//     PlcTask Inputs/GVL_iXlinker.EtherCAT_Master_EPPxxxx.Beckhoff_EPP6xxx.Beckhoff_EPP6xxxEK1122.A_0009_EPP6228_0022_0016.Module_1_DeviceState_Inputs_Device.DeviceState_Inputs_Device.Device_State <-> Module 1 (DeviceState Inputs Device)/DeviceState Inputs Device/Device State
//     PlcTask Inputs/GVL_iXlinker.EtherCAT_Master_EPPxxxx.Beckhoff_EPP6xxx.Beckhoff_EPP6xxxEK1122.A_0009_EPP6228_0022_0016.Module_2_DeviceState_Inputs.DeviceState_Inputs.State_Ch1 <-> Module 2 (DeviceState Inputs)/DeviceState Inputs/State Ch1
//     PlcTask Inputs/GVL_iXlinker.EtherCAT_Master_EPPxxxx.Beckhoff_EPP6xxx.Beckhoff_EPP6xxxEK1122.A_0009_EPP6228_0022_0016.Module_2_DeviceState_Inputs.DeviceState_Inputs.State_Ch2 <-> Module 2 (DeviceState Inputs)/DeviceState Inputs/State Ch2
//     PlcTask Inputs/GVL_iXlinker.EtherCAT_Master_EPPxxxx.Beckhoff_EPP6xxx.Beckhoff_EPP6xxxEK1122.A_0009_EPP6228_0022_0016.Module_2_DeviceState_Inputs.DeviceState_Inputs.State_Ch3 <-> Module 2 (DeviceState Inputs)/DeviceState Inputs/State Ch3
//     PlcTask Inputs/GVL_iXlinker.EtherCAT_Master_EPPxxxx.Beckhoff_EPP6xxx.Beckhoff_EPP6xxxEK1122.A_0009_EPP6228_0022_0016.Module_2_DeviceState_Inputs.DeviceState_Inputs.State_Ch4 <-> Module 2 (DeviceState Inputs)/DeviceState Inputs/State Ch4
//     PlcTask Inputs/GVL_iXlinker.EtherCAT_Master_EPPxxxx.Beckhoff_EPP6xxx.Beckhoff_EPP6xxxEK1122.A_0009_EPP6228_0022_0016.Module_2_DeviceState_Inputs.DeviceState_Inputs.State_Ch5 <-> Module 2 (DeviceState Inputs)/DeviceState Inputs/State Ch5
//     PlcTask Inputs/GVL_iXlinker.EtherCAT_Master_EPPxxxx.Beckhoff_EPP6xxx.Beckhoff_EPP6xxxEK1122.A_0009_EPP6228_0022_0016.Module_2_DeviceState_Inputs.DeviceState_Inputs.State_Ch6 <-> Module 2 (DeviceState Inputs)/DeviceState Inputs/State Ch6
//     PlcTask Inputs/GVL_iXlinker.EtherCAT_Master_EPPxxxx.Beckhoff_EPP6xxx.Beckhoff_EPP6xxxEK1122.A_0009_EPP6228_0022_0016.Module_2_DeviceState_Inputs.DeviceState_Inputs.State_Ch7 <-> Module 2 (DeviceState Inputs)/DeviceState Inputs/State Ch7
//     PlcTask Inputs/GVL_iXlinker.EtherCAT_Master_EPPxxxx.Beckhoff_EPP6xxx.Beckhoff_EPP6xxxEK1122.A_0009_EPP6228_0022_0016.Module_2_DeviceState_Inputs.DeviceState_Inputs.State_Ch8 <-> Module 2 (DeviceState Inputs)/DeviceState Inputs/State Ch8
//     PlcTask Inputs/GVL_iXlinker.EtherCAT_Master_EPPxxxx.Beckhoff_EPP6xxx.Beckhoff_EPP6xxxEK1122.A_0009_EPP6228_0022_0016.Module_11_Digital_Inputs.Digital_Inputs.Pin2_Ch1 <-> Module 11 (Digital Inputs)/Digital Inputs/Pin2 Ch1
//     PlcTask Inputs/GVL_iXlinker.EtherCAT_Master_EPPxxxx.Beckhoff_EPP6xxx.Beckhoff_EPP6xxxEK1122.A_0009_EPP6228_0022_0016.Module_11_Digital_Inputs.Digital_Inputs.Pin2_Ch2 <-> Module 11 (Digital Inputs)/Digital Inputs/Pin2 Ch2
//     PlcTask Inputs/GVL_iXlinker.EtherCAT_Master_EPPxxxx.Beckhoff_EPP6xxx.Beckhoff_EPP6xxxEK1122.A_0009_EPP6228_0022_0016.Module_11_Digital_Inputs.Digital_Inputs.Pin2_Ch3 <-> Module 11 (Digital Inputs)/Digital Inputs/Pin2 Ch3
//     PlcTask Inputs/GVL_iXlinker.EtherCAT_Master_EPPxxxx.Beckhoff_EPP6xxx.Beckhoff_EPP6xxxEK1122.A_0009_EPP6228_0022_0016.Module_11_Digital_Inputs.Digital_Inputs.Pin2_Ch4 <-> Module 11 (Digital Inputs)/Digital Inputs/Pin2 Ch4
//     PlcTask Inputs/GVL_iXlinker.EtherCAT_Master_EPPxxxx.Beckhoff_EPP6xxx.Beckhoff_EPP6xxxEK1122.A_0009_EPP6228_0022_0016.Module_11_Digital_Inputs.Digital_Inputs.Pin2_Ch5 <-> Module 11 (Digital Inputs)/Digital Inputs/Pin2 Ch5
//     PlcTask Inputs/GVL_iXlinker.EtherCAT_Master_EPPxxxx.Beckhoff_EPP6xxx.Beckhoff_EPP6xxxEK1122.A_0009_EPP6228_0022_0016.Module_11_Digital_Inputs.Digital_Inputs.Pin2_Ch6 <-> Module 11 (Digital Inputs)/Digital Inputs/Pin2 Ch6
//     PlcTask Inputs/GVL_iXlinker.EtherCAT_Master_EPPxxxx.Beckhoff_EPP6xxx.Beckhoff_EPP6xxxEK1122.A_0009_EPP6228_0022_0016.Module_11_Digital_Inputs.Digital_Inputs.Pin2_Ch7 <-> Module 11 (Digital Inputs)/Digital Inputs/Pin2 Ch7
//     PlcTask Inputs/GVL_iXlinker.EtherCAT_Master_EPPxxxx.Beckhoff_EPP6xxx.Beckhoff_EPP6xxxEK1122.A_0009_EPP6228_0022_0016.Module_11_Digital_Inputs.Digital_Inputs.Pin2_Ch8 <-> Module 11 (Digital Inputs)/Digital Inputs/Pin2 Ch8
//     PlcTask Inputs/GVL_iXlinker.EtherCAT_Master_EPPxxxx.Beckhoff_EPP6xxx.Beckhoff_EPP6xxxEK1122.A_0009_EPP6228_0022_0016.WcState.WcState <-> WcState/WcState
//     PlcTask Inputs/GVL_iXlinker.EtherCAT_Master_EPPxxxx.Beckhoff_EPP6xxx.Beckhoff_EPP6xxxEK1122.A_0009_EPP6228_0022_0016.WcState.InputToggle <-> WcState/InputToggle
//     PlcTask Inputs/GVL_iXlinker.EtherCAT_Master_EPPxxxx.Beckhoff_EPP6xxx.Beckhoff_EPP6xxxEK1122.A_0009_EPP6228_0022_0016.InfoData.AdsAddr <-> InfoData/AdsAddr
//     PlcTask Inputs/GVL_iXlinker.EtherCAT_Master_EPPxxxx.Beckhoff_EPP6xxx.Beckhoff_EPP6xxxEK1122.A_0009_EPP6228_0022_0016.InfoData.AoeNetId <-> InfoData/AoeNetId
//     PlcTask Inputs/GVL_iXlinker.EtherCAT_Master_EPPxxxx.Beckhoff_EPP6xxx.Beckhoff_EPP6xxxEK1122.A_0009_EPP6228_0022_0016.InfoData.State <-> InfoData/State
//   PLC/PLC Instance <-> EtherCAT Master EPPxxxx/Beckhoff EPP7xxx
//     PlcTask Inputs/GVL_iXlinker.EtherCAT_Master_EPPxxxx.Beckhoff_EPP7xxx.InfoData.State <-> InfoData/State
//   PLC/PLC Instance <-> EtherCAT Master EPPxxxx/Beckhoff EPP7xxx/Beckhoff EPP7xxxEK1122
//     PlcTask Inputs/GVL_iXlinker.EtherCAT_Master_EPPxxxx.Beckhoff_EPP7xxx.Beckhoff_EPP7xxxEK1122.InfoData.State <-> InfoData/State
//   PLC/PLC Instance <-> EtherCAT Master EPPxxxx/Beckhoff EPP7xxx/Beckhoff EPP7xxxEK1122/Beckhoff EPP7xxxsub EK1100
//     PlcTask Inputs/GVL_iXlinker.EtherCAT_Master_EPPxxxx.Beckhoff_EPP7xxx.Beckhoff_EPP7xxxEK1122.Beckhoff_EPP7xxxsub_EK1100.InfoData.State <-> InfoData/State
//   PLC/PLC Instance <-> EtherCAT Master EPPxxxx/Beckhoff EPP7xxx/Beckhoff EPP7xxxEK1122/A_0001(EPP7041-1002-0016)
//     PlcTask Inputs/GVL_iXlinker.EtherCAT_Master_EPPxxxx.Beckhoff_EPP7xxx.Beckhoff_EPP7xxxEK1122.A_0001_EPP7041_1002_0016.ENC_Status_compact.Status/Latch_C_valid <-> ENC Status compact/Status/Latch C valid
//     PlcTask Inputs/GVL_iXlinker.EtherCAT_Master_EPPxxxx.Beckhoff_EPP7xxx.Beckhoff_EPP7xxxEK1122.A_0001_EPP7041_1002_0016.ENC_Status_compact.Status/Latch_extern_valid <-> ENC Status compact/Status/Latch extern valid
//     PlcTask Inputs/GVL_iXlinker.EtherCAT_Master_EPPxxxx.Beckhoff_EPP7xxx.Beckhoff_EPP7xxxEK1122.A_0001_EPP7041_1002_0016.ENC_Status_compact.Status/Set_counter_done <-> ENC Status compact/Status/Set counter done
//     PlcTask Inputs/GVL_iXlinker.EtherCAT_Master_EPPxxxx.Beckhoff_EPP7xxx.Beckhoff_EPP7xxxEK1122.A_0001_EPP7041_1002_0016.ENC_Status_compact.Status/Counter_underflow <-> ENC Status compact/Status/Counter underflow
//     PlcTask Inputs/GVL_iXlinker.EtherCAT_Master_EPPxxxx.Beckhoff_EPP7xxx.Beckhoff_EPP7xxxEK1122.A_0001_EPP7041_1002_0016.ENC_Status_compact.Status/Counter_overflow <-> ENC Status compact/Status/Counter overflow
//     PlcTask Inputs/GVL_iXlinker.EtherCAT_Master_EPPxxxx.Beckhoff_EPP7xxx.Beckhoff_EPP7xxxEK1122.A_0001_EPP7041_1002_0016.ENC_Status_compact.Status/Extrapolation_stall <-> ENC Status compact/Status/Extrapolation stall
//     PlcTask Inputs/GVL_iXlinker.EtherCAT_Master_EPPxxxx.Beckhoff_EPP7xxx.Beckhoff_EPP7xxxEK1122.A_0001_EPP7041_1002_0016.ENC_Status_compact.Status/Status_of_input_A <-> ENC Status compact/Status/Status of input A
//     PlcTask Inputs/GVL_iXlinker.EtherCAT_Master_EPPxxxx.Beckhoff_EPP7xxx.Beckhoff_EPP7xxxEK1122.A_0001_EPP7041_1002_0016.ENC_Status_compact.Status/Status_of_input_B <-> ENC Status compact/Status/Status of input B
//     PlcTask Inputs/GVL_iXlinker.EtherCAT_Master_EPPxxxx.Beckhoff_EPP7xxx.Beckhoff_EPP7xxxEK1122.A_0001_EPP7041_1002_0016.ENC_Status_compact.Status/Status_of_input_C <-> ENC Status compact/Status/Status of input C
//     PlcTask Inputs/GVL_iXlinker.EtherCAT_Master_EPPxxxx.Beckhoff_EPP7xxx.Beckhoff_EPP7xxxEK1122.A_0001_EPP7041_1002_0016.ENC_Status_compact.Status/Status_of_extern_latch <-> ENC Status compact/Status/Status of extern latch
//     PlcTask Inputs/GVL_iXlinker.EtherCAT_Master_EPPxxxx.Beckhoff_EPP7xxx.Beckhoff_EPP7xxxEK1122.A_0001_EPP7041_1002_0016.ENC_Status_compact.Status/Sync_error <-> ENC Status compact/Status/Sync error
//     PlcTask Inputs/GVL_iXlinker.EtherCAT_Master_EPPxxxx.Beckhoff_EPP7xxx.Beckhoff_EPP7xxxEK1122.A_0001_EPP7041_1002_0016.ENC_Status_compact.Status/TxPDO_Toggle <-> ENC Status compact/Status/TxPDO Toggle
//     PlcTask Inputs/GVL_iXlinker.EtherCAT_Master_EPPxxxx.Beckhoff_EPP7xxx.Beckhoff_EPP7xxxEK1122.A_0001_EPP7041_1002_0016.ENC_Status_compact.Counter_value <-> ENC Status compact/Counter value
//     PlcTask Inputs/GVL_iXlinker.EtherCAT_Master_EPPxxxx.Beckhoff_EPP7xxx.Beckhoff_EPP7xxxEK1122.A_0001_EPP7041_1002_0016.ENC_Status_compact.Latch_value <-> ENC Status compact/Latch value
//     PlcTask Inputs/GVL_iXlinker.EtherCAT_Master_EPPxxxx.Beckhoff_EPP7xxx.Beckhoff_EPP7xxxEK1122.A_0001_EPP7041_1002_0016.STM_Status.Status/Ready_to_enable <-> STM Status/Status/Ready to enable
//     PlcTask Inputs/GVL_iXlinker.EtherCAT_Master_EPPxxxx.Beckhoff_EPP7xxx.Beckhoff_EPP7xxxEK1122.A_0001_EPP7041_1002_0016.STM_Status.Status/Ready <-> STM Status/Status/Ready
//     PlcTask Inputs/GVL_iXlinker.EtherCAT_Master_EPPxxxx.Beckhoff_EPP7xxx.Beckhoff_EPP7xxxEK1122.A_0001_EPP7041_1002_0016.STM_Status.Status/Warning <-> STM Status/Status/Warning
//     PlcTask Inputs/GVL_iXlinker.EtherCAT_Master_EPPxxxx.Beckhoff_EPP7xxx.Beckhoff_EPP7xxxEK1122.A_0001_EPP7041_1002_0016.STM_Status.Status/Error <-> STM Status/Status/Error
//     PlcTask Inputs/GVL_iXlinker.EtherCAT_Master_EPPxxxx.Beckhoff_EPP7xxx.Beckhoff_EPP7xxxEK1122.A_0001_EPP7041_1002_0016.STM_Status.Status/Moving_positive <-> STM Status/Status/Moving positive
//     PlcTask Inputs/GVL_iXlinker.EtherCAT_Master_EPPxxxx.Beckhoff_EPP7xxx.Beckhoff_EPP7xxxEK1122.A_0001_EPP7041_1002_0016.STM_Status.Status/Moving_negative <-> STM Status/Status/Moving negative
//     PlcTask Inputs/GVL_iXlinker.EtherCAT_Master_EPPxxxx.Beckhoff_EPP7xxx.Beckhoff_EPP7xxxEK1122.A_0001_EPP7041_1002_0016.STM_Status.Status/Torque_reduced <-> STM Status/Status/Torque reduced
//     PlcTask Inputs/GVL_iXlinker.EtherCAT_Master_EPPxxxx.Beckhoff_EPP7xxx.Beckhoff_EPP7xxxEK1122.A_0001_EPP7041_1002_0016.STM_Status.Status/Digital_input_1 <-> STM Status/Status/Digital input 1
//     PlcTask Inputs/GVL_iXlinker.EtherCAT_Master_EPPxxxx.Beckhoff_EPP7xxx.Beckhoff_EPP7xxxEK1122.A_0001_EPP7041_1002_0016.STM_Status.Status/Digital_input_2 <-> STM Status/Status/Digital input 2
//     PlcTask Inputs/GVL_iXlinker.EtherCAT_Master_EPPxxxx.Beckhoff_EPP7xxx.Beckhoff_EPP7xxxEK1122.A_0001_EPP7041_1002_0016.STM_Status.Status/Sync_error <-> STM Status/Status/Sync error
//     PlcTask Inputs/GVL_iXlinker.EtherCAT_Master_EPPxxxx.Beckhoff_EPP7xxx.Beckhoff_EPP7xxxEK1122.A_0001_EPP7041_1002_0016.STM_Status.Status/TxPDO_Toggle <-> STM Status/Status/TxPDO Toggle
//     PlcTask Outputs/GVL_iXlinker.EtherCAT_Master_EPPxxxx.Beckhoff_EPP7xxx.Beckhoff_EPP7xxxEK1122.A_0001_EPP7041_1002_0016.ENC_Control_compact.Control/Enable_latch_C <-> ENC Control compact/Control/Enable latch C
//     PlcTask Outputs/GVL_iXlinker.EtherCAT_Master_EPPxxxx.Beckhoff_EPP7xxx.Beckhoff_EPP7xxxEK1122.A_0001_EPP7041_1002_0016.ENC_Control_compact.Control/Enable_latch_extern_on_positive_edge <-> ENC Control compact/Control/Enable latch extern on positive edge
//     PlcTask Outputs/GVL_iXlinker.EtherCAT_Master_EPPxxxx.Beckhoff_EPP7xxx.Beckhoff_EPP7xxxEK1122.A_0001_EPP7041_1002_0016.ENC_Control_compact.Control/Set_counter <-> ENC Control compact/Control/Set counter
//     PlcTask Outputs/GVL_iXlinker.EtherCAT_Master_EPPxxxx.Beckhoff_EPP7xxx.Beckhoff_EPP7xxxEK1122.A_0001_EPP7041_1002_0016.ENC_Control_compact.Control/Enable_latch_extern_on_negative_edge <-> ENC Control compact/Control/Enable latch extern on negative edge
//     PlcTask Outputs/GVL_iXlinker.EtherCAT_Master_EPPxxxx.Beckhoff_EPP7xxx.Beckhoff_EPP7xxxEK1122.A_0001_EPP7041_1002_0016.ENC_Control_compact.Set_counter_value <-> ENC Control compact/Set counter value
//     PlcTask Outputs/GVL_iXlinker.EtherCAT_Master_EPPxxxx.Beckhoff_EPP7xxx.Beckhoff_EPP7xxxEK1122.A_0001_EPP7041_1002_0016.STM_Control.Control/Enable <-> STM Control/Control/Enable
//     PlcTask Outputs/GVL_iXlinker.EtherCAT_Master_EPPxxxx.Beckhoff_EPP7xxx.Beckhoff_EPP7xxxEK1122.A_0001_EPP7041_1002_0016.STM_Control.Control/Reset <-> STM Control/Control/Reset
//     PlcTask Outputs/GVL_iXlinker.EtherCAT_Master_EPPxxxx.Beckhoff_EPP7xxx.Beckhoff_EPP7xxxEK1122.A_0001_EPP7041_1002_0016.STM_Control.Control/Reduce_torque <-> STM Control/Control/Reduce torque
//     PlcTask Outputs/GVL_iXlinker.EtherCAT_Master_EPPxxxx.Beckhoff_EPP7xxx.Beckhoff_EPP7xxxEK1122.A_0001_EPP7041_1002_0016.STM_Control.Control/Digital_output_1 <-> STM Control/Control/Digital output 1
//     PlcTask Outputs/GVL_iXlinker.EtherCAT_Master_EPPxxxx.Beckhoff_EPP7xxx.Beckhoff_EPP7xxxEK1122.A_0001_EPP7041_1002_0016.STM_Velocity.Velocity <-> STM Velocity/Velocity
//     PlcTask Inputs/GVL_iXlinker.EtherCAT_Master_EPPxxxx.Beckhoff_EPP7xxx.Beckhoff_EPP7xxxEK1122.A_0001_EPP7041_1002_0016.WcState.WcState <-> WcState/WcState
//     PlcTask Inputs/GVL_iXlinker.EtherCAT_Master_EPPxxxx.Beckhoff_EPP7xxx.Beckhoff_EPP7xxxEK1122.A_0001_EPP7041_1002_0016.WcState.InputToggle <-> WcState/InputToggle
//     PlcTask Inputs/GVL_iXlinker.EtherCAT_Master_EPPxxxx.Beckhoff_EPP7xxx.Beckhoff_EPP7xxxEK1122.A_0001_EPP7041_1002_0016.InfoData.AdsAddr <-> InfoData/AdsAddr
//     PlcTask Inputs/GVL_iXlinker.EtherCAT_Master_EPPxxxx.Beckhoff_EPP7xxx.Beckhoff_EPP7xxxEK1122.A_0001_EPP7041_1002_0016.InfoData.Chn0 <-> InfoData/Chn0
//     PlcTask Inputs/GVL_iXlinker.EtherCAT_Master_EPPxxxx.Beckhoff_EPP7xxx.Beckhoff_EPP7xxxEK1122.A_0001_EPP7041_1002_0016.InfoData.Chn1 <-> InfoData/Chn1
//     PlcTask Inputs/GVL_iXlinker.EtherCAT_Master_EPPxxxx.Beckhoff_EPP7xxx.Beckhoff_EPP7xxxEK1122.A_0001_EPP7041_1002_0016.InfoData.State <-> InfoData/State
//   PLC/PLC Instance <-> EtherCAT Master EPPxxxx/Beckhoff EPP7xxx/Beckhoff EPP7xxxEK1122/A_0002(EPP7041-1002-0017)
//     PlcTask Inputs/GVL_iXlinker.EtherCAT_Master_EPPxxxx.Beckhoff_EPP7xxx.Beckhoff_EPP7xxxEK1122.A_0002_EPP7041_1002_0017.ENC_Status_compact.Status/Latch_C_valid <-> ENC Status compact/Status/Latch C valid
//     PlcTask Inputs/GVL_iXlinker.EtherCAT_Master_EPPxxxx.Beckhoff_EPP7xxx.Beckhoff_EPP7xxxEK1122.A_0002_EPP7041_1002_0017.ENC_Status_compact.Status/Latch_extern_valid <-> ENC Status compact/Status/Latch extern valid
//     PlcTask Inputs/GVL_iXlinker.EtherCAT_Master_EPPxxxx.Beckhoff_EPP7xxx.Beckhoff_EPP7xxxEK1122.A_0002_EPP7041_1002_0017.ENC_Status_compact.Status/Set_counter_done <-> ENC Status compact/Status/Set counter done
//     PlcTask Inputs/GVL_iXlinker.EtherCAT_Master_EPPxxxx.Beckhoff_EPP7xxx.Beckhoff_EPP7xxxEK1122.A_0002_EPP7041_1002_0017.ENC_Status_compact.Status/Counter_underflow <-> ENC Status compact/Status/Counter underflow
//     PlcTask Inputs/GVL_iXlinker.EtherCAT_Master_EPPxxxx.Beckhoff_EPP7xxx.Beckhoff_EPP7xxxEK1122.A_0002_EPP7041_1002_0017.ENC_Status_compact.Status/Counter_overflow <-> ENC Status compact/Status/Counter overflow
//     PlcTask Inputs/GVL_iXlinker.EtherCAT_Master_EPPxxxx.Beckhoff_EPP7xxx.Beckhoff_EPP7xxxEK1122.A_0002_EPP7041_1002_0017.ENC_Status_compact.Status/Extrapolation_stall <-> ENC Status compact/Status/Extrapolation stall
//     PlcTask Inputs/GVL_iXlinker.EtherCAT_Master_EPPxxxx.Beckhoff_EPP7xxx.Beckhoff_EPP7xxxEK1122.A_0002_EPP7041_1002_0017.ENC_Status_compact.Status/Status_of_input_A <-> ENC Status compact/Status/Status of input A
//     PlcTask Inputs/GVL_iXlinker.EtherCAT_Master_EPPxxxx.Beckhoff_EPP7xxx.Beckhoff_EPP7xxxEK1122.A_0002_EPP7041_1002_0017.ENC_Status_compact.Status/Status_of_input_B <-> ENC Status compact/Status/Status of input B
//     PlcTask Inputs/GVL_iXlinker.EtherCAT_Master_EPPxxxx.Beckhoff_EPP7xxx.Beckhoff_EPP7xxxEK1122.A_0002_EPP7041_1002_0017.ENC_Status_compact.Status/Status_of_input_C <-> ENC Status compact/Status/Status of input C
//     PlcTask Inputs/GVL_iXlinker.EtherCAT_Master_EPPxxxx.Beckhoff_EPP7xxx.Beckhoff_EPP7xxxEK1122.A_0002_EPP7041_1002_0017.ENC_Status_compact.Status/Status_of_extern_latch <-> ENC Status compact/Status/Status of extern latch
//     PlcTask Inputs/GVL_iXlinker.EtherCAT_Master_EPPxxxx.Beckhoff_EPP7xxx.Beckhoff_EPP7xxxEK1122.A_0002_EPP7041_1002_0017.ENC_Status_compact.Status/Sync_error <-> ENC Status compact/Status/Sync error
//     PlcTask Inputs/GVL_iXlinker.EtherCAT_Master_EPPxxxx.Beckhoff_EPP7xxx.Beckhoff_EPP7xxxEK1122.A_0002_EPP7041_1002_0017.ENC_Status_compact.Status/TxPDO_Toggle <-> ENC Status compact/Status/TxPDO Toggle
//     PlcTask Inputs/GVL_iXlinker.EtherCAT_Master_EPPxxxx.Beckhoff_EPP7xxx.Beckhoff_EPP7xxxEK1122.A_0002_EPP7041_1002_0017.ENC_Status_compact.Counter_value <-> ENC Status compact/Counter value
//     PlcTask Inputs/GVL_iXlinker.EtherCAT_Master_EPPxxxx.Beckhoff_EPP7xxx.Beckhoff_EPP7xxxEK1122.A_0002_EPP7041_1002_0017.ENC_Status_compact.Latch_value <-> ENC Status compact/Latch value
//     PlcTask Inputs/GVL_iXlinker.EtherCAT_Master_EPPxxxx.Beckhoff_EPP7xxx.Beckhoff_EPP7xxxEK1122.A_0002_EPP7041_1002_0017.STM_Status.Status/Ready_to_enable <-> STM Status/Status/Ready to enable
//     PlcTask Inputs/GVL_iXlinker.EtherCAT_Master_EPPxxxx.Beckhoff_EPP7xxx.Beckhoff_EPP7xxxEK1122.A_0002_EPP7041_1002_0017.STM_Status.Status/Ready <-> STM Status/Status/Ready
//     PlcTask Inputs/GVL_iXlinker.EtherCAT_Master_EPPxxxx.Beckhoff_EPP7xxx.Beckhoff_EPP7xxxEK1122.A_0002_EPP7041_1002_0017.STM_Status.Status/Warning <-> STM Status/Status/Warning
//     PlcTask Inputs/GVL_iXlinker.EtherCAT_Master_EPPxxxx.Beckhoff_EPP7xxx.Beckhoff_EPP7xxxEK1122.A_0002_EPP7041_1002_0017.STM_Status.Status/Error <-> STM Status/Status/Error
//     PlcTask Inputs/GVL_iXlinker.EtherCAT_Master_EPPxxxx.Beckhoff_EPP7xxx.Beckhoff_EPP7xxxEK1122.A_0002_EPP7041_1002_0017.STM_Status.Status/Moving_positive <-> STM Status/Status/Moving positive
//     PlcTask Inputs/GVL_iXlinker.EtherCAT_Master_EPPxxxx.Beckhoff_EPP7xxx.Beckhoff_EPP7xxxEK1122.A_0002_EPP7041_1002_0017.STM_Status.Status/Moving_negative <-> STM Status/Status/Moving negative
//     PlcTask Inputs/GVL_iXlinker.EtherCAT_Master_EPPxxxx.Beckhoff_EPP7xxx.Beckhoff_EPP7xxxEK1122.A_0002_EPP7041_1002_0017.STM_Status.Status/Torque_reduced <-> STM Status/Status/Torque reduced
//     PlcTask Inputs/GVL_iXlinker.EtherCAT_Master_EPPxxxx.Beckhoff_EPP7xxx.Beckhoff_EPP7xxxEK1122.A_0002_EPP7041_1002_0017.STM_Status.Status/Digital_input_1 <-> STM Status/Status/Digital input 1
//     PlcTask Inputs/GVL_iXlinker.EtherCAT_Master_EPPxxxx.Beckhoff_EPP7xxx.Beckhoff_EPP7xxxEK1122.A_0002_EPP7041_1002_0017.STM_Status.Status/Digital_input_2 <-> STM Status/Status/Digital input 2
//     PlcTask Inputs/GVL_iXlinker.EtherCAT_Master_EPPxxxx.Beckhoff_EPP7xxx.Beckhoff_EPP7xxxEK1122.A_0002_EPP7041_1002_0017.STM_Status.Status/Sync_error <-> STM Status/Status/Sync error
//     PlcTask Inputs/GVL_iXlinker.EtherCAT_Master_EPPxxxx.Beckhoff_EPP7xxx.Beckhoff_EPP7xxxEK1122.A_0002_EPP7041_1002_0017.STM_Status.Status/TxPDO_Toggle <-> STM Status/Status/TxPDO Toggle
//     PlcTask Outputs/GVL_iXlinker.EtherCAT_Master_EPPxxxx.Beckhoff_EPP7xxx.Beckhoff_EPP7xxxEK1122.A_0002_EPP7041_1002_0017.ENC_Control_compact.Control/Enable_latch_C <-> ENC Control compact/Control/Enable latch C
//     PlcTask Outputs/GVL_iXlinker.EtherCAT_Master_EPPxxxx.Beckhoff_EPP7xxx.Beckhoff_EPP7xxxEK1122.A_0002_EPP7041_1002_0017.ENC_Control_compact.Control/Enable_latch_extern_on_positive_edge <-> ENC Control compact/Control/Enable latch extern on positive edge
//     PlcTask Outputs/GVL_iXlinker.EtherCAT_Master_EPPxxxx.Beckhoff_EPP7xxx.Beckhoff_EPP7xxxEK1122.A_0002_EPP7041_1002_0017.ENC_Control_compact.Control/Set_counter <-> ENC Control compact/Control/Set counter
//     PlcTask Outputs/GVL_iXlinker.EtherCAT_Master_EPPxxxx.Beckhoff_EPP7xxx.Beckhoff_EPP7xxxEK1122.A_0002_EPP7041_1002_0017.ENC_Control_compact.Control/Enable_latch_extern_on_negative_edge <-> ENC Control compact/Control/Enable latch extern on negative edge
//     PlcTask Outputs/GVL_iXlinker.EtherCAT_Master_EPPxxxx.Beckhoff_EPP7xxx.Beckhoff_EPP7xxxEK1122.A_0002_EPP7041_1002_0017.ENC_Control_compact.Set_counter_value <-> ENC Control compact/Set counter value
//     PlcTask Outputs/GVL_iXlinker.EtherCAT_Master_EPPxxxx.Beckhoff_EPP7xxx.Beckhoff_EPP7xxxEK1122.A_0002_EPP7041_1002_0017.STM_Control.Control/Enable <-> STM Control/Control/Enable
//     PlcTask Outputs/GVL_iXlinker.EtherCAT_Master_EPPxxxx.Beckhoff_EPP7xxx.Beckhoff_EPP7xxxEK1122.A_0002_EPP7041_1002_0017.STM_Control.Control/Reset <-> STM Control/Control/Reset
//     PlcTask Outputs/GVL_iXlinker.EtherCAT_Master_EPPxxxx.Beckhoff_EPP7xxx.Beckhoff_EPP7xxxEK1122.A_0002_EPP7041_1002_0017.STM_Control.Control/Reduce_torque <-> STM Control/Control/Reduce torque
//     PlcTask Outputs/GVL_iXlinker.EtherCAT_Master_EPPxxxx.Beckhoff_EPP7xxx.Beckhoff_EPP7xxxEK1122.A_0002_EPP7041_1002_0017.STM_Control.Control/Digital_output_1 <-> STM Control/Control/Digital output 1
//     PlcTask Outputs/GVL_iXlinker.EtherCAT_Master_EPPxxxx.Beckhoff_EPP7xxx.Beckhoff_EPP7xxxEK1122.A_0002_EPP7041_1002_0017.STM_Velocity.Velocity <-> STM Velocity/Velocity
//     PlcTask Inputs/GVL_iXlinker.EtherCAT_Master_EPPxxxx.Beckhoff_EPP7xxx.Beckhoff_EPP7xxxEK1122.A_0002_EPP7041_1002_0017.WcState.WcState <-> WcState/WcState
//     PlcTask Inputs/GVL_iXlinker.EtherCAT_Master_EPPxxxx.Beckhoff_EPP7xxx.Beckhoff_EPP7xxxEK1122.A_0002_EPP7041_1002_0017.WcState.InputToggle <-> WcState/InputToggle
//     PlcTask Inputs/GVL_iXlinker.EtherCAT_Master_EPPxxxx.Beckhoff_EPP7xxx.Beckhoff_EPP7xxxEK1122.A_0002_EPP7041_1002_0017.InfoData.AdsAddr <-> InfoData/AdsAddr
//     PlcTask Inputs/GVL_iXlinker.EtherCAT_Master_EPPxxxx.Beckhoff_EPP7xxx.Beckhoff_EPP7xxxEK1122.A_0002_EPP7041_1002_0017.InfoData.Chn0 <-> InfoData/Chn0
//     PlcTask Inputs/GVL_iXlinker.EtherCAT_Master_EPPxxxx.Beckhoff_EPP7xxx.Beckhoff_EPP7xxxEK1122.A_0002_EPP7041_1002_0017.InfoData.Chn1 <-> InfoData/Chn1
//     PlcTask Inputs/GVL_iXlinker.EtherCAT_Master_EPPxxxx.Beckhoff_EPP7xxx.Beckhoff_EPP7xxxEK1122.A_0002_EPP7041_1002_0017.InfoData.State <-> InfoData/State
//   PLC/PLC Instance <-> EtherCAT Master EPPxxxx/Beckhoff EPP7xxx/Beckhoff EPP7xxxEK1122/A_0003(EPP7041-1002-0023)
//     PlcTask Inputs/GVL_iXlinker.EtherCAT_Master_EPPxxxx.Beckhoff_EPP7xxx.Beckhoff_EPP7xxxEK1122.A_0003_EPP7041_1002_0023.ENC_Status_compact.Status/Latch_C_valid <-> ENC Status compact/Status/Latch C valid
//     PlcTask Inputs/GVL_iXlinker.EtherCAT_Master_EPPxxxx.Beckhoff_EPP7xxx.Beckhoff_EPP7xxxEK1122.A_0003_EPP7041_1002_0023.ENC_Status_compact.Status/Latch_extern_valid <-> ENC Status compact/Status/Latch extern valid
//     PlcTask Inputs/GVL_iXlinker.EtherCAT_Master_EPPxxxx.Beckhoff_EPP7xxx.Beckhoff_EPP7xxxEK1122.A_0003_EPP7041_1002_0023.ENC_Status_compact.Status/Set_counter_done <-> ENC Status compact/Status/Set counter done
//     PlcTask Inputs/GVL_iXlinker.EtherCAT_Master_EPPxxxx.Beckhoff_EPP7xxx.Beckhoff_EPP7xxxEK1122.A_0003_EPP7041_1002_0023.ENC_Status_compact.Status/Counter_underflow <-> ENC Status compact/Status/Counter underflow
//     PlcTask Inputs/GVL_iXlinker.EtherCAT_Master_EPPxxxx.Beckhoff_EPP7xxx.Beckhoff_EPP7xxxEK1122.A_0003_EPP7041_1002_0023.ENC_Status_compact.Status/Counter_overflow <-> ENC Status compact/Status/Counter overflow
//     PlcTask Inputs/GVL_iXlinker.EtherCAT_Master_EPPxxxx.Beckhoff_EPP7xxx.Beckhoff_EPP7xxxEK1122.A_0003_EPP7041_1002_0023.ENC_Status_compact.Status/Extrapolation_stall <-> ENC Status compact/Status/Extrapolation stall
//     PlcTask Inputs/GVL_iXlinker.EtherCAT_Master_EPPxxxx.Beckhoff_EPP7xxx.Beckhoff_EPP7xxxEK1122.A_0003_EPP7041_1002_0023.ENC_Status_compact.Status/Status_of_input_A <-> ENC Status compact/Status/Status of input A
//     PlcTask Inputs/GVL_iXlinker.EtherCAT_Master_EPPxxxx.Beckhoff_EPP7xxx.Beckhoff_EPP7xxxEK1122.A_0003_EPP7041_1002_0023.ENC_Status_compact.Status/Status_of_input_B <-> ENC Status compact/Status/Status of input B
//     PlcTask Inputs/GVL_iXlinker.EtherCAT_Master_EPPxxxx.Beckhoff_EPP7xxx.Beckhoff_EPP7xxxEK1122.A_0003_EPP7041_1002_0023.ENC_Status_compact.Status/Status_of_input_C <-> ENC Status compact/Status/Status of input C
//     PlcTask Inputs/GVL_iXlinker.EtherCAT_Master_EPPxxxx.Beckhoff_EPP7xxx.Beckhoff_EPP7xxxEK1122.A_0003_EPP7041_1002_0023.ENC_Status_compact.Status/Status_of_extern_latch <-> ENC Status compact/Status/Status of extern latch
//     PlcTask Inputs/GVL_iXlinker.EtherCAT_Master_EPPxxxx.Beckhoff_EPP7xxx.Beckhoff_EPP7xxxEK1122.A_0003_EPP7041_1002_0023.ENC_Status_compact.Status/Sync_error <-> ENC Status compact/Status/Sync error
//     PlcTask Inputs/GVL_iXlinker.EtherCAT_Master_EPPxxxx.Beckhoff_EPP7xxx.Beckhoff_EPP7xxxEK1122.A_0003_EPP7041_1002_0023.ENC_Status_compact.Status/TxPDO_Toggle <-> ENC Status compact/Status/TxPDO Toggle
//     PlcTask Inputs/GVL_iXlinker.EtherCAT_Master_EPPxxxx.Beckhoff_EPP7xxx.Beckhoff_EPP7xxxEK1122.A_0003_EPP7041_1002_0023.ENC_Status_compact.Counter_value <-> ENC Status compact/Counter value
//     PlcTask Inputs/GVL_iXlinker.EtherCAT_Master_EPPxxxx.Beckhoff_EPP7xxx.Beckhoff_EPP7xxxEK1122.A_0003_EPP7041_1002_0023.ENC_Status_compact.Latch_value <-> ENC Status compact/Latch value
//     PlcTask Inputs/GVL_iXlinker.EtherCAT_Master_EPPxxxx.Beckhoff_EPP7xxx.Beckhoff_EPP7xxxEK1122.A_0003_EPP7041_1002_0023.STM_Status.Status/Ready_to_enable <-> STM Status/Status/Ready to enable
//     PlcTask Inputs/GVL_iXlinker.EtherCAT_Master_EPPxxxx.Beckhoff_EPP7xxx.Beckhoff_EPP7xxxEK1122.A_0003_EPP7041_1002_0023.STM_Status.Status/Ready <-> STM Status/Status/Ready
//     PlcTask Inputs/GVL_iXlinker.EtherCAT_Master_EPPxxxx.Beckhoff_EPP7xxx.Beckhoff_EPP7xxxEK1122.A_0003_EPP7041_1002_0023.STM_Status.Status/Warning <-> STM Status/Status/Warning
//     PlcTask Inputs/GVL_iXlinker.EtherCAT_Master_EPPxxxx.Beckhoff_EPP7xxx.Beckhoff_EPP7xxxEK1122.A_0003_EPP7041_1002_0023.STM_Status.Status/Error <-> STM Status/Status/Error
//     PlcTask Inputs/GVL_iXlinker.EtherCAT_Master_EPPxxxx.Beckhoff_EPP7xxx.Beckhoff_EPP7xxxEK1122.A_0003_EPP7041_1002_0023.STM_Status.Status/Moving_positive <-> STM Status/Status/Moving positive
//     PlcTask Inputs/GVL_iXlinker.EtherCAT_Master_EPPxxxx.Beckhoff_EPP7xxx.Beckhoff_EPP7xxxEK1122.A_0003_EPP7041_1002_0023.STM_Status.Status/Moving_negative <-> STM Status/Status/Moving negative
//     PlcTask Inputs/GVL_iXlinker.EtherCAT_Master_EPPxxxx.Beckhoff_EPP7xxx.Beckhoff_EPP7xxxEK1122.A_0003_EPP7041_1002_0023.STM_Status.Status/Torque_reduced <-> STM Status/Status/Torque reduced
//     PlcTask Inputs/GVL_iXlinker.EtherCAT_Master_EPPxxxx.Beckhoff_EPP7xxx.Beckhoff_EPP7xxxEK1122.A_0003_EPP7041_1002_0023.STM_Status.Status/Motor_stall <-> STM Status/Status/Motor stall
//     PlcTask Inputs/GVL_iXlinker.EtherCAT_Master_EPPxxxx.Beckhoff_EPP7xxx.Beckhoff_EPP7xxxEK1122.A_0003_EPP7041_1002_0023.STM_Status.Status/Digital_input_1 <-> STM Status/Status/Digital input 1
//     PlcTask Inputs/GVL_iXlinker.EtherCAT_Master_EPPxxxx.Beckhoff_EPP7xxx.Beckhoff_EPP7xxxEK1122.A_0003_EPP7041_1002_0023.STM_Status.Status/Digital_input_2 <-> STM Status/Status/Digital input 2
//     PlcTask Inputs/GVL_iXlinker.EtherCAT_Master_EPPxxxx.Beckhoff_EPP7xxx.Beckhoff_EPP7xxxEK1122.A_0003_EPP7041_1002_0023.STM_Status.Status/Sync_error <-> STM Status/Status/Sync error
//     PlcTask Inputs/GVL_iXlinker.EtherCAT_Master_EPPxxxx.Beckhoff_EPP7xxx.Beckhoff_EPP7xxxEK1122.A_0003_EPP7041_1002_0023.STM_Status.Status/TxPDO_Toggle <-> STM Status/Status/TxPDO Toggle
//     PlcTask Outputs/GVL_iXlinker.EtherCAT_Master_EPPxxxx.Beckhoff_EPP7xxx.Beckhoff_EPP7xxxEK1122.A_0003_EPP7041_1002_0023.ENC_Control_compact.Control/Enable_latch_C <-> ENC Control compact/Control/Enable latch C
//     PlcTask Outputs/GVL_iXlinker.EtherCAT_Master_EPPxxxx.Beckhoff_EPP7xxx.Beckhoff_EPP7xxxEK1122.A_0003_EPP7041_1002_0023.ENC_Control_compact.Control/Enable_latch_extern_on_positive_edge <-> ENC Control compact/Control/Enable latch extern on positive edge
//     PlcTask Outputs/GVL_iXlinker.EtherCAT_Master_EPPxxxx.Beckhoff_EPP7xxx.Beckhoff_EPP7xxxEK1122.A_0003_EPP7041_1002_0023.ENC_Control_compact.Control/Set_counter <-> ENC Control compact/Control/Set counter
//     PlcTask Outputs/GVL_iXlinker.EtherCAT_Master_EPPxxxx.Beckhoff_EPP7xxx.Beckhoff_EPP7xxxEK1122.A_0003_EPP7041_1002_0023.ENC_Control_compact.Control/Enable_latch_extern_on_negative_edge <-> ENC Control compact/Control/Enable latch extern on negative edge
//     PlcTask Outputs/GVL_iXlinker.EtherCAT_Master_EPPxxxx.Beckhoff_EPP7xxx.Beckhoff_EPP7xxxEK1122.A_0003_EPP7041_1002_0023.ENC_Control_compact.Set_counter_value <-> ENC Control compact/Set counter value
//     PlcTask Outputs/GVL_iXlinker.EtherCAT_Master_EPPxxxx.Beckhoff_EPP7xxx.Beckhoff_EPP7xxxEK1122.A_0003_EPP7041_1002_0023.STM_Control.Control/Enable <-> STM Control/Control/Enable
//     PlcTask Outputs/GVL_iXlinker.EtherCAT_Master_EPPxxxx.Beckhoff_EPP7xxx.Beckhoff_EPP7xxxEK1122.A_0003_EPP7041_1002_0023.STM_Control.Control/Reset <-> STM Control/Control/Reset
//     PlcTask Outputs/GVL_iXlinker.EtherCAT_Master_EPPxxxx.Beckhoff_EPP7xxx.Beckhoff_EPP7xxxEK1122.A_0003_EPP7041_1002_0023.STM_Control.Control/Reduce_torque <-> STM Control/Control/Reduce torque
//     PlcTask Outputs/GVL_iXlinker.EtherCAT_Master_EPPxxxx.Beckhoff_EPP7xxx.Beckhoff_EPP7xxxEK1122.A_0003_EPP7041_1002_0023.STM_Control.Control/Digital_output_1 <-> STM Control/Control/Digital output 1
//     PlcTask Outputs/GVL_iXlinker.EtherCAT_Master_EPPxxxx.Beckhoff_EPP7xxx.Beckhoff_EPP7xxxEK1122.A_0003_EPP7041_1002_0023.STM_Velocity.Velocity <-> STM Velocity/Velocity
//     PlcTask Inputs/GVL_iXlinker.EtherCAT_Master_EPPxxxx.Beckhoff_EPP7xxx.Beckhoff_EPP7xxxEK1122.A_0003_EPP7041_1002_0023.WcState.WcState <-> WcState/WcState
//     PlcTask Inputs/GVL_iXlinker.EtherCAT_Master_EPPxxxx.Beckhoff_EPP7xxx.Beckhoff_EPP7xxxEK1122.A_0003_EPP7041_1002_0023.WcState.InputToggle <-> WcState/InputToggle
//     PlcTask Inputs/GVL_iXlinker.EtherCAT_Master_EPPxxxx.Beckhoff_EPP7xxx.Beckhoff_EPP7xxxEK1122.A_0003_EPP7041_1002_0023.InfoData.AdsAddr <-> InfoData/AdsAddr
//     PlcTask Inputs/GVL_iXlinker.EtherCAT_Master_EPPxxxx.Beckhoff_EPP7xxx.Beckhoff_EPP7xxxEK1122.A_0003_EPP7041_1002_0023.InfoData.Chn0 <-> InfoData/Chn0
//     PlcTask Inputs/GVL_iXlinker.EtherCAT_Master_EPPxxxx.Beckhoff_EPP7xxx.Beckhoff_EPP7xxxEK1122.A_0003_EPP7041_1002_0023.InfoData.Chn1 <-> InfoData/Chn1
//     PlcTask Inputs/GVL_iXlinker.EtherCAT_Master_EPPxxxx.Beckhoff_EPP7xxx.Beckhoff_EPP7xxxEK1122.A_0003_EPP7041_1002_0023.InfoData.State <-> InfoData/State
//   PLC/PLC Instance <-> EtherCAT Master EPPxxxx/Beckhoff EPP7xxx/Beckhoff EPP7xxxEK1122/A_0004(EPP7041-3002-0016)
//     PlcTask Inputs/GVL_iXlinker.EtherCAT_Master_EPPxxxx.Beckhoff_EPP7xxx.Beckhoff_EPP7xxxEK1122.A_0004_EPP7041_3002_0016.ENC_Status_compact.Status/Latch_C_valid <-> ENC Status compact/Status/Latch C valid
//     PlcTask Inputs/GVL_iXlinker.EtherCAT_Master_EPPxxxx.Beckhoff_EPP7xxx.Beckhoff_EPP7xxxEK1122.A_0004_EPP7041_3002_0016.ENC_Status_compact.Status/Latch_extern_valid <-> ENC Status compact/Status/Latch extern valid
//     PlcTask Inputs/GVL_iXlinker.EtherCAT_Master_EPPxxxx.Beckhoff_EPP7xxx.Beckhoff_EPP7xxxEK1122.A_0004_EPP7041_3002_0016.ENC_Status_compact.Status/Set_counter_done <-> ENC Status compact/Status/Set counter done
//     PlcTask Inputs/GVL_iXlinker.EtherCAT_Master_EPPxxxx.Beckhoff_EPP7xxx.Beckhoff_EPP7xxxEK1122.A_0004_EPP7041_3002_0016.ENC_Status_compact.Status/Counter_underflow <-> ENC Status compact/Status/Counter underflow
//     PlcTask Inputs/GVL_iXlinker.EtherCAT_Master_EPPxxxx.Beckhoff_EPP7xxx.Beckhoff_EPP7xxxEK1122.A_0004_EPP7041_3002_0016.ENC_Status_compact.Status/Counter_overflow <-> ENC Status compact/Status/Counter overflow
//     PlcTask Inputs/GVL_iXlinker.EtherCAT_Master_EPPxxxx.Beckhoff_EPP7xxx.Beckhoff_EPP7xxxEK1122.A_0004_EPP7041_3002_0016.ENC_Status_compact.Status/Extrapolation_stall <-> ENC Status compact/Status/Extrapolation stall
//     PlcTask Inputs/GVL_iXlinker.EtherCAT_Master_EPPxxxx.Beckhoff_EPP7xxx.Beckhoff_EPP7xxxEK1122.A_0004_EPP7041_3002_0016.ENC_Status_compact.Status/Status_of_input_A <-> ENC Status compact/Status/Status of input A
//     PlcTask Inputs/GVL_iXlinker.EtherCAT_Master_EPPxxxx.Beckhoff_EPP7xxx.Beckhoff_EPP7xxxEK1122.A_0004_EPP7041_3002_0016.ENC_Status_compact.Status/Status_of_input_B <-> ENC Status compact/Status/Status of input B
//     PlcTask Inputs/GVL_iXlinker.EtherCAT_Master_EPPxxxx.Beckhoff_EPP7xxx.Beckhoff_EPP7xxxEK1122.A_0004_EPP7041_3002_0016.ENC_Status_compact.Status/Status_of_input_C <-> ENC Status compact/Status/Status of input C
//     PlcTask Inputs/GVL_iXlinker.EtherCAT_Master_EPPxxxx.Beckhoff_EPP7xxx.Beckhoff_EPP7xxxEK1122.A_0004_EPP7041_3002_0016.ENC_Status_compact.Status/Status_of_extern_latch <-> ENC Status compact/Status/Status of extern latch
//     PlcTask Inputs/GVL_iXlinker.EtherCAT_Master_EPPxxxx.Beckhoff_EPP7xxx.Beckhoff_EPP7xxxEK1122.A_0004_EPP7041_3002_0016.ENC_Status_compact.Status/Sync_error <-> ENC Status compact/Status/Sync error
//     PlcTask Inputs/GVL_iXlinker.EtherCAT_Master_EPPxxxx.Beckhoff_EPP7xxx.Beckhoff_EPP7xxxEK1122.A_0004_EPP7041_3002_0016.ENC_Status_compact.Status/TxPDO_Toggle <-> ENC Status compact/Status/TxPDO Toggle
//     PlcTask Inputs/GVL_iXlinker.EtherCAT_Master_EPPxxxx.Beckhoff_EPP7xxx.Beckhoff_EPP7xxxEK1122.A_0004_EPP7041_3002_0016.ENC_Status_compact.Counter_value <-> ENC Status compact/Counter value
//     PlcTask Inputs/GVL_iXlinker.EtherCAT_Master_EPPxxxx.Beckhoff_EPP7xxx.Beckhoff_EPP7xxxEK1122.A_0004_EPP7041_3002_0016.ENC_Status_compact.Latch_value <-> ENC Status compact/Latch value
//     PlcTask Inputs/GVL_iXlinker.EtherCAT_Master_EPPxxxx.Beckhoff_EPP7xxx.Beckhoff_EPP7xxxEK1122.A_0004_EPP7041_3002_0016.STM_Status.Status/Ready_to_enable <-> STM Status/Status/Ready to enable
//     PlcTask Inputs/GVL_iXlinker.EtherCAT_Master_EPPxxxx.Beckhoff_EPP7xxx.Beckhoff_EPP7xxxEK1122.A_0004_EPP7041_3002_0016.STM_Status.Status/Ready <-> STM Status/Status/Ready
//     PlcTask Inputs/GVL_iXlinker.EtherCAT_Master_EPPxxxx.Beckhoff_EPP7xxx.Beckhoff_EPP7xxxEK1122.A_0004_EPP7041_3002_0016.STM_Status.Status/Warning <-> STM Status/Status/Warning
//     PlcTask Inputs/GVL_iXlinker.EtherCAT_Master_EPPxxxx.Beckhoff_EPP7xxx.Beckhoff_EPP7xxxEK1122.A_0004_EPP7041_3002_0016.STM_Status.Status/Error <-> STM Status/Status/Error
//     PlcTask Inputs/GVL_iXlinker.EtherCAT_Master_EPPxxxx.Beckhoff_EPP7xxx.Beckhoff_EPP7xxxEK1122.A_0004_EPP7041_3002_0016.STM_Status.Status/Moving_positive <-> STM Status/Status/Moving positive
//     PlcTask Inputs/GVL_iXlinker.EtherCAT_Master_EPPxxxx.Beckhoff_EPP7xxx.Beckhoff_EPP7xxxEK1122.A_0004_EPP7041_3002_0016.STM_Status.Status/Moving_negative <-> STM Status/Status/Moving negative
//     PlcTask Inputs/GVL_iXlinker.EtherCAT_Master_EPPxxxx.Beckhoff_EPP7xxx.Beckhoff_EPP7xxxEK1122.A_0004_EPP7041_3002_0016.STM_Status.Status/Torque_reduced <-> STM Status/Status/Torque reduced
//     PlcTask Inputs/GVL_iXlinker.EtherCAT_Master_EPPxxxx.Beckhoff_EPP7xxx.Beckhoff_EPP7xxxEK1122.A_0004_EPP7041_3002_0016.STM_Status.Status/Motor_stall <-> STM Status/Status/Motor stall
//     PlcTask Inputs/GVL_iXlinker.EtherCAT_Master_EPPxxxx.Beckhoff_EPP7xxx.Beckhoff_EPP7xxxEK1122.A_0004_EPP7041_3002_0016.STM_Status.Status/Digital_input_1 <-> STM Status/Status/Digital input 1
//     PlcTask Inputs/GVL_iXlinker.EtherCAT_Master_EPPxxxx.Beckhoff_EPP7xxx.Beckhoff_EPP7xxxEK1122.A_0004_EPP7041_3002_0016.STM_Status.Status/Digital_input_2 <-> STM Status/Status/Digital input 2
//     PlcTask Inputs/GVL_iXlinker.EtherCAT_Master_EPPxxxx.Beckhoff_EPP7xxx.Beckhoff_EPP7xxxEK1122.A_0004_EPP7041_3002_0016.STM_Status.Status/Sync_error <-> STM Status/Status/Sync error
//     PlcTask Inputs/GVL_iXlinker.EtherCAT_Master_EPPxxxx.Beckhoff_EPP7xxx.Beckhoff_EPP7xxxEK1122.A_0004_EPP7041_3002_0016.STM_Status.Status/TxPDO_Toggle <-> STM Status/Status/TxPDO Toggle
//     PlcTask Outputs/GVL_iXlinker.EtherCAT_Master_EPPxxxx.Beckhoff_EPP7xxx.Beckhoff_EPP7xxxEK1122.A_0004_EPP7041_3002_0016.ENC_Control_compact.Control/Enable_latch_C <-> ENC Control compact/Control/Enable latch C
//     PlcTask Outputs/GVL_iXlinker.EtherCAT_Master_EPPxxxx.Beckhoff_EPP7xxx.Beckhoff_EPP7xxxEK1122.A_0004_EPP7041_3002_0016.ENC_Control_compact.Control/Enable_latch_extern_on_positive_edge <-> ENC Control compact/Control/Enable latch extern on positive edge
//     PlcTask Outputs/GVL_iXlinker.EtherCAT_Master_EPPxxxx.Beckhoff_EPP7xxx.Beckhoff_EPP7xxxEK1122.A_0004_EPP7041_3002_0016.ENC_Control_compact.Control/Set_counter <-> ENC Control compact/Control/Set counter
//     PlcTask Outputs/GVL_iXlinker.EtherCAT_Master_EPPxxxx.Beckhoff_EPP7xxx.Beckhoff_EPP7xxxEK1122.A_0004_EPP7041_3002_0016.ENC_Control_compact.Control/Enable_latch_extern_on_negative_edge <-> ENC Control compact/Control/Enable latch extern on negative edge
//     PlcTask Outputs/GVL_iXlinker.EtherCAT_Master_EPPxxxx.Beckhoff_EPP7xxx.Beckhoff_EPP7xxxEK1122.A_0004_EPP7041_3002_0016.ENC_Control_compact.Set_counter_value <-> ENC Control compact/Set counter value
//     PlcTask Outputs/GVL_iXlinker.EtherCAT_Master_EPPxxxx.Beckhoff_EPP7xxx.Beckhoff_EPP7xxxEK1122.A_0004_EPP7041_3002_0016.STM_Control.Control/Enable <-> STM Control/Control/Enable
//     PlcTask Outputs/GVL_iXlinker.EtherCAT_Master_EPPxxxx.Beckhoff_EPP7xxx.Beckhoff_EPP7xxxEK1122.A_0004_EPP7041_3002_0016.STM_Control.Control/Reset <-> STM Control/Control/Reset
//     PlcTask Outputs/GVL_iXlinker.EtherCAT_Master_EPPxxxx.Beckhoff_EPP7xxx.Beckhoff_EPP7xxxEK1122.A_0004_EPP7041_3002_0016.STM_Control.Control/Reduce_torque <-> STM Control/Control/Reduce torque
//     PlcTask Outputs/GVL_iXlinker.EtherCAT_Master_EPPxxxx.Beckhoff_EPP7xxx.Beckhoff_EPP7xxxEK1122.A_0004_EPP7041_3002_0016.STM_Control.Control/Digital_output_1 <-> STM Control/Control/Digital output 1
//     PlcTask Outputs/GVL_iXlinker.EtherCAT_Master_EPPxxxx.Beckhoff_EPP7xxx.Beckhoff_EPP7xxxEK1122.A_0004_EPP7041_3002_0016.STM_Velocity.Velocity <-> STM Velocity/Velocity
//     PlcTask Inputs/GVL_iXlinker.EtherCAT_Master_EPPxxxx.Beckhoff_EPP7xxx.Beckhoff_EPP7xxxEK1122.A_0004_EPP7041_3002_0016.WcState.WcState <-> WcState/WcState
//     PlcTask Inputs/GVL_iXlinker.EtherCAT_Master_EPPxxxx.Beckhoff_EPP7xxx.Beckhoff_EPP7xxxEK1122.A_0004_EPP7041_3002_0016.WcState.InputToggle <-> WcState/InputToggle
//     PlcTask Inputs/GVL_iXlinker.EtherCAT_Master_EPPxxxx.Beckhoff_EPP7xxx.Beckhoff_EPP7xxxEK1122.A_0004_EPP7041_3002_0016.InfoData.AdsAddr <-> InfoData/AdsAddr
//     PlcTask Inputs/GVL_iXlinker.EtherCAT_Master_EPPxxxx.Beckhoff_EPP7xxx.Beckhoff_EPP7xxxEK1122.A_0004_EPP7041_3002_0016.InfoData.Chn0 <-> InfoData/Chn0
//     PlcTask Inputs/GVL_iXlinker.EtherCAT_Master_EPPxxxx.Beckhoff_EPP7xxx.Beckhoff_EPP7xxxEK1122.A_0004_EPP7041_3002_0016.InfoData.Chn1 <-> InfoData/Chn1
//     PlcTask Inputs/GVL_iXlinker.EtherCAT_Master_EPPxxxx.Beckhoff_EPP7xxx.Beckhoff_EPP7xxxEK1122.A_0004_EPP7041_3002_0016.InfoData.State <-> InfoData/State
//   PLC/PLC Instance <-> EtherCAT Master EPPxxxx/Beckhoff EPP7xxx/Beckhoff EPP7xxxEK1122/A_0005(EPP7041-3002-0017)
//     PlcTask Inputs/GVL_iXlinker.EtherCAT_Master_EPPxxxx.Beckhoff_EPP7xxx.Beckhoff_EPP7xxxEK1122.A_0005_EPP7041_3002_0017.ENC_Status_compact.Status/Latch_C_valid <-> ENC Status compact/Status/Latch C valid
//     PlcTask Inputs/GVL_iXlinker.EtherCAT_Master_EPPxxxx.Beckhoff_EPP7xxx.Beckhoff_EPP7xxxEK1122.A_0005_EPP7041_3002_0017.ENC_Status_compact.Status/Latch_extern_valid <-> ENC Status compact/Status/Latch extern valid
//     PlcTask Inputs/GVL_iXlinker.EtherCAT_Master_EPPxxxx.Beckhoff_EPP7xxx.Beckhoff_EPP7xxxEK1122.A_0005_EPP7041_3002_0017.ENC_Status_compact.Status/Set_counter_done <-> ENC Status compact/Status/Set counter done
//     PlcTask Inputs/GVL_iXlinker.EtherCAT_Master_EPPxxxx.Beckhoff_EPP7xxx.Beckhoff_EPP7xxxEK1122.A_0005_EPP7041_3002_0017.ENC_Status_compact.Status/Counter_underflow <-> ENC Status compact/Status/Counter underflow
//     PlcTask Inputs/GVL_iXlinker.EtherCAT_Master_EPPxxxx.Beckhoff_EPP7xxx.Beckhoff_EPP7xxxEK1122.A_0005_EPP7041_3002_0017.ENC_Status_compact.Status/Counter_overflow <-> ENC Status compact/Status/Counter overflow
//     PlcTask Inputs/GVL_iXlinker.EtherCAT_Master_EPPxxxx.Beckhoff_EPP7xxx.Beckhoff_EPP7xxxEK1122.A_0005_EPP7041_3002_0017.ENC_Status_compact.Status/Extrapolation_stall <-> ENC Status compact/Status/Extrapolation stall
//     PlcTask Inputs/GVL_iXlinker.EtherCAT_Master_EPPxxxx.Beckhoff_EPP7xxx.Beckhoff_EPP7xxxEK1122.A_0005_EPP7041_3002_0017.ENC_Status_compact.Status/Status_of_input_A <-> ENC Status compact/Status/Status of input A
//     PlcTask Inputs/GVL_iXlinker.EtherCAT_Master_EPPxxxx.Beckhoff_EPP7xxx.Beckhoff_EPP7xxxEK1122.A_0005_EPP7041_3002_0017.ENC_Status_compact.Status/Status_of_input_B <-> ENC Status compact/Status/Status of input B
//     PlcTask Inputs/GVL_iXlinker.EtherCAT_Master_EPPxxxx.Beckhoff_EPP7xxx.Beckhoff_EPP7xxxEK1122.A_0005_EPP7041_3002_0017.ENC_Status_compact.Status/Status_of_input_C <-> ENC Status compact/Status/Status of input C
//     PlcTask Inputs/GVL_iXlinker.EtherCAT_Master_EPPxxxx.Beckhoff_EPP7xxx.Beckhoff_EPP7xxxEK1122.A_0005_EPP7041_3002_0017.ENC_Status_compact.Status/Status_of_extern_latch <-> ENC Status compact/Status/Status of extern latch
//     PlcTask Inputs/GVL_iXlinker.EtherCAT_Master_EPPxxxx.Beckhoff_EPP7xxx.Beckhoff_EPP7xxxEK1122.A_0005_EPP7041_3002_0017.ENC_Status_compact.Status/Sync_error <-> ENC Status compact/Status/Sync error
//     PlcTask Inputs/GVL_iXlinker.EtherCAT_Master_EPPxxxx.Beckhoff_EPP7xxx.Beckhoff_EPP7xxxEK1122.A_0005_EPP7041_3002_0017.ENC_Status_compact.Status/TxPDO_Toggle <-> ENC Status compact/Status/TxPDO Toggle
//     PlcTask Inputs/GVL_iXlinker.EtherCAT_Master_EPPxxxx.Beckhoff_EPP7xxx.Beckhoff_EPP7xxxEK1122.A_0005_EPP7041_3002_0017.ENC_Status_compact.Counter_value <-> ENC Status compact/Counter value
//     PlcTask Inputs/GVL_iXlinker.EtherCAT_Master_EPPxxxx.Beckhoff_EPP7xxx.Beckhoff_EPP7xxxEK1122.A_0005_EPP7041_3002_0017.ENC_Status_compact.Latch_value <-> ENC Status compact/Latch value
//     PlcTask Inputs/GVL_iXlinker.EtherCAT_Master_EPPxxxx.Beckhoff_EPP7xxx.Beckhoff_EPP7xxxEK1122.A_0005_EPP7041_3002_0017.STM_Status.Status/Ready_to_enable <-> STM Status/Status/Ready to enable
//     PlcTask Inputs/GVL_iXlinker.EtherCAT_Master_EPPxxxx.Beckhoff_EPP7xxx.Beckhoff_EPP7xxxEK1122.A_0005_EPP7041_3002_0017.STM_Status.Status/Ready <-> STM Status/Status/Ready
//     PlcTask Inputs/GVL_iXlinker.EtherCAT_Master_EPPxxxx.Beckhoff_EPP7xxx.Beckhoff_EPP7xxxEK1122.A_0005_EPP7041_3002_0017.STM_Status.Status/Warning <-> STM Status/Status/Warning
//     PlcTask Inputs/GVL_iXlinker.EtherCAT_Master_EPPxxxx.Beckhoff_EPP7xxx.Beckhoff_EPP7xxxEK1122.A_0005_EPP7041_3002_0017.STM_Status.Status/Error <-> STM Status/Status/Error
//     PlcTask Inputs/GVL_iXlinker.EtherCAT_Master_EPPxxxx.Beckhoff_EPP7xxx.Beckhoff_EPP7xxxEK1122.A_0005_EPP7041_3002_0017.STM_Status.Status/Moving_positive <-> STM Status/Status/Moving positive
//     PlcTask Inputs/GVL_iXlinker.EtherCAT_Master_EPPxxxx.Beckhoff_EPP7xxx.Beckhoff_EPP7xxxEK1122.A_0005_EPP7041_3002_0017.STM_Status.Status/Moving_negative <-> STM Status/Status/Moving negative
//     PlcTask Inputs/GVL_iXlinker.EtherCAT_Master_EPPxxxx.Beckhoff_EPP7xxx.Beckhoff_EPP7xxxEK1122.A_0005_EPP7041_3002_0017.STM_Status.Status/Torque_reduced <-> STM Status/Status/Torque reduced
//     PlcTask Inputs/GVL_iXlinker.EtherCAT_Master_EPPxxxx.Beckhoff_EPP7xxx.Beckhoff_EPP7xxxEK1122.A_0005_EPP7041_3002_0017.STM_Status.Status/Motor_stall <-> STM Status/Status/Motor stall
//     PlcTask Inputs/GVL_iXlinker.EtherCAT_Master_EPPxxxx.Beckhoff_EPP7xxx.Beckhoff_EPP7xxxEK1122.A_0005_EPP7041_3002_0017.STM_Status.Status/Digital_input_1 <-> STM Status/Status/Digital input 1
//     PlcTask Inputs/GVL_iXlinker.EtherCAT_Master_EPPxxxx.Beckhoff_EPP7xxx.Beckhoff_EPP7xxxEK1122.A_0005_EPP7041_3002_0017.STM_Status.Status/Digital_input_2 <-> STM Status/Status/Digital input 2
//     PlcTask Inputs/GVL_iXlinker.EtherCAT_Master_EPPxxxx.Beckhoff_EPP7xxx.Beckhoff_EPP7xxxEK1122.A_0005_EPP7041_3002_0017.STM_Status.Status/Sync_error <-> STM Status/Status/Sync error
//     PlcTask Inputs/GVL_iXlinker.EtherCAT_Master_EPPxxxx.Beckhoff_EPP7xxx.Beckhoff_EPP7xxxEK1122.A_0005_EPP7041_3002_0017.STM_Status.Status/TxPDO_Toggle <-> STM Status/Status/TxPDO Toggle
//     PlcTask Outputs/GVL_iXlinker.EtherCAT_Master_EPPxxxx.Beckhoff_EPP7xxx.Beckhoff_EPP7xxxEK1122.A_0005_EPP7041_3002_0017.ENC_Control_compact.Control/Enable_latch_C <-> ENC Control compact/Control/Enable latch C
//     PlcTask Outputs/GVL_iXlinker.EtherCAT_Master_EPPxxxx.Beckhoff_EPP7xxx.Beckhoff_EPP7xxxEK1122.A_0005_EPP7041_3002_0017.ENC_Control_compact.Control/Enable_latch_extern_on_positive_edge <-> ENC Control compact/Control/Enable latch extern on positive edge
//     PlcTask Outputs/GVL_iXlinker.EtherCAT_Master_EPPxxxx.Beckhoff_EPP7xxx.Beckhoff_EPP7xxxEK1122.A_0005_EPP7041_3002_0017.ENC_Control_compact.Control/Set_counter <-> ENC Control compact/Control/Set counter
//     PlcTask Outputs/GVL_iXlinker.EtherCAT_Master_EPPxxxx.Beckhoff_EPP7xxx.Beckhoff_EPP7xxxEK1122.A_0005_EPP7041_3002_0017.ENC_Control_compact.Control/Enable_latch_extern_on_negative_edge <-> ENC Control compact/Control/Enable latch extern on negative edge
//     PlcTask Outputs/GVL_iXlinker.EtherCAT_Master_EPPxxxx.Beckhoff_EPP7xxx.Beckhoff_EPP7xxxEK1122.A_0005_EPP7041_3002_0017.ENC_Control_compact.Set_counter_value <-> ENC Control compact/Set counter value
//     PlcTask Outputs/GVL_iXlinker.EtherCAT_Master_EPPxxxx.Beckhoff_EPP7xxx.Beckhoff_EPP7xxxEK1122.A_0005_EPP7041_3002_0017.STM_Control.Control/Enable <-> STM Control/Control/Enable
//     PlcTask Outputs/GVL_iXlinker.EtherCAT_Master_EPPxxxx.Beckhoff_EPP7xxx.Beckhoff_EPP7xxxEK1122.A_0005_EPP7041_3002_0017.STM_Control.Control/Reset <-> STM Control/Control/Reset
//     PlcTask Outputs/GVL_iXlinker.EtherCAT_Master_EPPxxxx.Beckhoff_EPP7xxx.Beckhoff_EPP7xxxEK1122.A_0005_EPP7041_3002_0017.STM_Control.Control/Reduce_torque <-> STM Control/Control/Reduce torque
//     PlcTask Outputs/GVL_iXlinker.EtherCAT_Master_EPPxxxx.Beckhoff_EPP7xxx.Beckhoff_EPP7xxxEK1122.A_0005_EPP7041_3002_0017.STM_Control.Control/Digital_output_1 <-> STM Control/Control/Digital output 1
//     PlcTask Outputs/GVL_iXlinker.EtherCAT_Master_EPPxxxx.Beckhoff_EPP7xxx.Beckhoff_EPP7xxxEK1122.A_0005_EPP7041_3002_0017.STM_Velocity.Velocity <-> STM Velocity/Velocity
//     PlcTask Inputs/GVL_iXlinker.EtherCAT_Master_EPPxxxx.Beckhoff_EPP7xxx.Beckhoff_EPP7xxxEK1122.A_0005_EPP7041_3002_0017.WcState.WcState <-> WcState/WcState
//     PlcTask Inputs/GVL_iXlinker.EtherCAT_Master_EPPxxxx.Beckhoff_EPP7xxx.Beckhoff_EPP7xxxEK1122.A_0005_EPP7041_3002_0017.WcState.InputToggle <-> WcState/InputToggle
//     PlcTask Inputs/GVL_iXlinker.EtherCAT_Master_EPPxxxx.Beckhoff_EPP7xxx.Beckhoff_EPP7xxxEK1122.A_0005_EPP7041_3002_0017.InfoData.AdsAddr <-> InfoData/AdsAddr
//     PlcTask Inputs/GVL_iXlinker.EtherCAT_Master_EPPxxxx.Beckhoff_EPP7xxx.Beckhoff_EPP7xxxEK1122.A_0005_EPP7041_3002_0017.InfoData.Chn0 <-> InfoData/Chn0
//     PlcTask Inputs/GVL_iXlinker.EtherCAT_Master_EPPxxxx.Beckhoff_EPP7xxx.Beckhoff_EPP7xxxEK1122.A_0005_EPP7041_3002_0017.InfoData.Chn1 <-> InfoData/Chn1
//     PlcTask Inputs/GVL_iXlinker.EtherCAT_Master_EPPxxxx.Beckhoff_EPP7xxx.Beckhoff_EPP7xxxEK1122.A_0005_EPP7041_3002_0017.InfoData.State <-> InfoData/State
//   PLC/PLC Instance <-> EtherCAT Master EPPxxxx/Beckhoff EPP7xxx/Beckhoff EPP7xxxEK1122/A_0006(EPP7041-3002-0018)
//     PlcTask Inputs/GVL_iXlinker.EtherCAT_Master_EPPxxxx.Beckhoff_EPP7xxx.Beckhoff_EPP7xxxEK1122.A_0006_EPP7041_3002_0018.ENC_Status_compact.Status/Latch_C_valid <-> ENC Status compact/Status/Latch C valid
//     PlcTask Inputs/GVL_iXlinker.EtherCAT_Master_EPPxxxx.Beckhoff_EPP7xxx.Beckhoff_EPP7xxxEK1122.A_0006_EPP7041_3002_0018.ENC_Status_compact.Status/Latch_extern_valid <-> ENC Status compact/Status/Latch extern valid
//     PlcTask Inputs/GVL_iXlinker.EtherCAT_Master_EPPxxxx.Beckhoff_EPP7xxx.Beckhoff_EPP7xxxEK1122.A_0006_EPP7041_3002_0018.ENC_Status_compact.Status/Set_counter_done <-> ENC Status compact/Status/Set counter done
//     PlcTask Inputs/GVL_iXlinker.EtherCAT_Master_EPPxxxx.Beckhoff_EPP7xxx.Beckhoff_EPP7xxxEK1122.A_0006_EPP7041_3002_0018.ENC_Status_compact.Status/Counter_underflow <-> ENC Status compact/Status/Counter underflow
//     PlcTask Inputs/GVL_iXlinker.EtherCAT_Master_EPPxxxx.Beckhoff_EPP7xxx.Beckhoff_EPP7xxxEK1122.A_0006_EPP7041_3002_0018.ENC_Status_compact.Status/Counter_overflow <-> ENC Status compact/Status/Counter overflow
//     PlcTask Inputs/GVL_iXlinker.EtherCAT_Master_EPPxxxx.Beckhoff_EPP7xxx.Beckhoff_EPP7xxxEK1122.A_0006_EPP7041_3002_0018.ENC_Status_compact.Status/Extrapolation_stall <-> ENC Status compact/Status/Extrapolation stall
//     PlcTask Inputs/GVL_iXlinker.EtherCAT_Master_EPPxxxx.Beckhoff_EPP7xxx.Beckhoff_EPP7xxxEK1122.A_0006_EPP7041_3002_0018.ENC_Status_compact.Status/Status_of_input_A <-> ENC Status compact/Status/Status of input A
//     PlcTask Inputs/GVL_iXlinker.EtherCAT_Master_EPPxxxx.Beckhoff_EPP7xxx.Beckhoff_EPP7xxxEK1122.A_0006_EPP7041_3002_0018.ENC_Status_compact.Status/Status_of_input_B <-> ENC Status compact/Status/Status of input B
//     PlcTask Inputs/GVL_iXlinker.EtherCAT_Master_EPPxxxx.Beckhoff_EPP7xxx.Beckhoff_EPP7xxxEK1122.A_0006_EPP7041_3002_0018.ENC_Status_compact.Status/Status_of_input_C <-> ENC Status compact/Status/Status of input C
//     PlcTask Inputs/GVL_iXlinker.EtherCAT_Master_EPPxxxx.Beckhoff_EPP7xxx.Beckhoff_EPP7xxxEK1122.A_0006_EPP7041_3002_0018.ENC_Status_compact.Status/Status_of_extern_latch <-> ENC Status compact/Status/Status of extern latch
//     PlcTask Inputs/GVL_iXlinker.EtherCAT_Master_EPPxxxx.Beckhoff_EPP7xxx.Beckhoff_EPP7xxxEK1122.A_0006_EPP7041_3002_0018.ENC_Status_compact.Status/Sync_error <-> ENC Status compact/Status/Sync error
//     PlcTask Inputs/GVL_iXlinker.EtherCAT_Master_EPPxxxx.Beckhoff_EPP7xxx.Beckhoff_EPP7xxxEK1122.A_0006_EPP7041_3002_0018.ENC_Status_compact.Status/TxPDO_Toggle <-> ENC Status compact/Status/TxPDO Toggle
//     PlcTask Inputs/GVL_iXlinker.EtherCAT_Master_EPPxxxx.Beckhoff_EPP7xxx.Beckhoff_EPP7xxxEK1122.A_0006_EPP7041_3002_0018.ENC_Status_compact.Counter_value <-> ENC Status compact/Counter value
//     PlcTask Inputs/GVL_iXlinker.EtherCAT_Master_EPPxxxx.Beckhoff_EPP7xxx.Beckhoff_EPP7xxxEK1122.A_0006_EPP7041_3002_0018.ENC_Status_compact.Latch_value <-> ENC Status compact/Latch value
//     PlcTask Inputs/GVL_iXlinker.EtherCAT_Master_EPPxxxx.Beckhoff_EPP7xxx.Beckhoff_EPP7xxxEK1122.A_0006_EPP7041_3002_0018.STM_Status.Status/Ready_to_enable <-> STM Status/Status/Ready to enable
//     PlcTask Inputs/GVL_iXlinker.EtherCAT_Master_EPPxxxx.Beckhoff_EPP7xxx.Beckhoff_EPP7xxxEK1122.A_0006_EPP7041_3002_0018.STM_Status.Status/Ready <-> STM Status/Status/Ready
//     PlcTask Inputs/GVL_iXlinker.EtherCAT_Master_EPPxxxx.Beckhoff_EPP7xxx.Beckhoff_EPP7xxxEK1122.A_0006_EPP7041_3002_0018.STM_Status.Status/Warning <-> STM Status/Status/Warning
//     PlcTask Inputs/GVL_iXlinker.EtherCAT_Master_EPPxxxx.Beckhoff_EPP7xxx.Beckhoff_EPP7xxxEK1122.A_0006_EPP7041_3002_0018.STM_Status.Status/Error <-> STM Status/Status/Error
//     PlcTask Inputs/GVL_iXlinker.EtherCAT_Master_EPPxxxx.Beckhoff_EPP7xxx.Beckhoff_EPP7xxxEK1122.A_0006_EPP7041_3002_0018.STM_Status.Status/Moving_positive <-> STM Status/Status/Moving positive
//     PlcTask Inputs/GVL_iXlinker.EtherCAT_Master_EPPxxxx.Beckhoff_EPP7xxx.Beckhoff_EPP7xxxEK1122.A_0006_EPP7041_3002_0018.STM_Status.Status/Moving_negative <-> STM Status/Status/Moving negative
//     PlcTask Inputs/GVL_iXlinker.EtherCAT_Master_EPPxxxx.Beckhoff_EPP7xxx.Beckhoff_EPP7xxxEK1122.A_0006_EPP7041_3002_0018.STM_Status.Status/Torque_reduced <-> STM Status/Status/Torque reduced
//     PlcTask Inputs/GVL_iXlinker.EtherCAT_Master_EPPxxxx.Beckhoff_EPP7xxx.Beckhoff_EPP7xxxEK1122.A_0006_EPP7041_3002_0018.STM_Status.Status/Motor_stall <-> STM Status/Status/Motor stall
//     PlcTask Inputs/GVL_iXlinker.EtherCAT_Master_EPPxxxx.Beckhoff_EPP7xxx.Beckhoff_EPP7xxxEK1122.A_0006_EPP7041_3002_0018.STM_Status.Status/Digital_input_1 <-> STM Status/Status/Digital input 1
//     PlcTask Inputs/GVL_iXlinker.EtherCAT_Master_EPPxxxx.Beckhoff_EPP7xxx.Beckhoff_EPP7xxxEK1122.A_0006_EPP7041_3002_0018.STM_Status.Status/Digital_input_2 <-> STM Status/Status/Digital input 2
//     PlcTask Inputs/GVL_iXlinker.EtherCAT_Master_EPPxxxx.Beckhoff_EPP7xxx.Beckhoff_EPP7xxxEK1122.A_0006_EPP7041_3002_0018.STM_Status.Status/Sync_error <-> STM Status/Status/Sync error
//     PlcTask Inputs/GVL_iXlinker.EtherCAT_Master_EPPxxxx.Beckhoff_EPP7xxx.Beckhoff_EPP7xxxEK1122.A_0006_EPP7041_3002_0018.STM_Status.Status/TxPDO_Toggle <-> STM Status/Status/TxPDO Toggle
//     PlcTask Outputs/GVL_iXlinker.EtherCAT_Master_EPPxxxx.Beckhoff_EPP7xxx.Beckhoff_EPP7xxxEK1122.A_0006_EPP7041_3002_0018.ENC_Control_compact.Control/Enable_latch_C <-> ENC Control compact/Control/Enable latch C
//     PlcTask Outputs/GVL_iXlinker.EtherCAT_Master_EPPxxxx.Beckhoff_EPP7xxx.Beckhoff_EPP7xxxEK1122.A_0006_EPP7041_3002_0018.ENC_Control_compact.Control/Enable_latch_extern_on_positive_edge <-> ENC Control compact/Control/Enable latch extern on positive edge
//     PlcTask Outputs/GVL_iXlinker.EtherCAT_Master_EPPxxxx.Beckhoff_EPP7xxx.Beckhoff_EPP7xxxEK1122.A_0006_EPP7041_3002_0018.ENC_Control_compact.Control/Set_counter <-> ENC Control compact/Control/Set counter
//     PlcTask Outputs/GVL_iXlinker.EtherCAT_Master_EPPxxxx.Beckhoff_EPP7xxx.Beckhoff_EPP7xxxEK1122.A_0006_EPP7041_3002_0018.ENC_Control_compact.Control/Enable_latch_extern_on_negative_edge <-> ENC Control compact/Control/Enable latch extern on negative edge
//     PlcTask Outputs/GVL_iXlinker.EtherCAT_Master_EPPxxxx.Beckhoff_EPP7xxx.Beckhoff_EPP7xxxEK1122.A_0006_EPP7041_3002_0018.ENC_Control_compact.Set_counter_value <-> ENC Control compact/Set counter value
//     PlcTask Outputs/GVL_iXlinker.EtherCAT_Master_EPPxxxx.Beckhoff_EPP7xxx.Beckhoff_EPP7xxxEK1122.A_0006_EPP7041_3002_0018.STM_Control.Control/Enable <-> STM Control/Control/Enable
//     PlcTask Outputs/GVL_iXlinker.EtherCAT_Master_EPPxxxx.Beckhoff_EPP7xxx.Beckhoff_EPP7xxxEK1122.A_0006_EPP7041_3002_0018.STM_Control.Control/Reset <-> STM Control/Control/Reset
//     PlcTask Outputs/GVL_iXlinker.EtherCAT_Master_EPPxxxx.Beckhoff_EPP7xxx.Beckhoff_EPP7xxxEK1122.A_0006_EPP7041_3002_0018.STM_Control.Control/Reduce_torque <-> STM Control/Control/Reduce torque
//     PlcTask Outputs/GVL_iXlinker.EtherCAT_Master_EPPxxxx.Beckhoff_EPP7xxx.Beckhoff_EPP7xxxEK1122.A_0006_EPP7041_3002_0018.STM_Control.Control/Digital_output_1 <-> STM Control/Control/Digital output 1
//     PlcTask Outputs/GVL_iXlinker.EtherCAT_Master_EPPxxxx.Beckhoff_EPP7xxx.Beckhoff_EPP7xxxEK1122.A_0006_EPP7041_3002_0018.STM_Velocity.Velocity <-> STM Velocity/Velocity
//     PlcTask Inputs/GVL_iXlinker.EtherCAT_Master_EPPxxxx.Beckhoff_EPP7xxx.Beckhoff_EPP7xxxEK1122.A_0006_EPP7041_3002_0018.WcState.WcState <-> WcState/WcState
//     PlcTask Inputs/GVL_iXlinker.EtherCAT_Master_EPPxxxx.Beckhoff_EPP7xxx.Beckhoff_EPP7xxxEK1122.A_0006_EPP7041_3002_0018.WcState.InputToggle <-> WcState/InputToggle
//     PlcTask Inputs/GVL_iXlinker.EtherCAT_Master_EPPxxxx.Beckhoff_EPP7xxx.Beckhoff_EPP7xxxEK1122.A_0006_EPP7041_3002_0018.InfoData.AdsAddr <-> InfoData/AdsAddr
//     PlcTask Inputs/GVL_iXlinker.EtherCAT_Master_EPPxxxx.Beckhoff_EPP7xxx.Beckhoff_EPP7xxxEK1122.A_0006_EPP7041_3002_0018.InfoData.Chn0 <-> InfoData/Chn0
//     PlcTask Inputs/GVL_iXlinker.EtherCAT_Master_EPPxxxx.Beckhoff_EPP7xxx.Beckhoff_EPP7xxxEK1122.A_0006_EPP7041_3002_0018.InfoData.Chn1 <-> InfoData/Chn1
//     PlcTask Inputs/GVL_iXlinker.EtherCAT_Master_EPPxxxx.Beckhoff_EPP7xxx.Beckhoff_EPP7xxxEK1122.A_0006_EPP7041_3002_0018.InfoData.State <-> InfoData/State
//   PLC/PLC Instance <-> EtherCAT Master EPPxxxx/Beckhoff EPP7xxx/Beckhoff EPP7xxxEK1122/A_0007(EPP7041-3002-0023)
//     PlcTask Inputs/GVL_iXlinker.EtherCAT_Master_EPPxxxx.Beckhoff_EPP7xxx.Beckhoff_EPP7xxxEK1122.A_0007_EPP7041_3002_0023.ENC_Status_compact.Status/Latch_C_valid <-> ENC Status compact/Status/Latch C valid
//     PlcTask Inputs/GVL_iXlinker.EtherCAT_Master_EPPxxxx.Beckhoff_EPP7xxx.Beckhoff_EPP7xxxEK1122.A_0007_EPP7041_3002_0023.ENC_Status_compact.Status/Latch_extern_valid <-> ENC Status compact/Status/Latch extern valid
//     PlcTask Inputs/GVL_iXlinker.EtherCAT_Master_EPPxxxx.Beckhoff_EPP7xxx.Beckhoff_EPP7xxxEK1122.A_0007_EPP7041_3002_0023.ENC_Status_compact.Status/Set_counter_done <-> ENC Status compact/Status/Set counter done
//     PlcTask Inputs/GVL_iXlinker.EtherCAT_Master_EPPxxxx.Beckhoff_EPP7xxx.Beckhoff_EPP7xxxEK1122.A_0007_EPP7041_3002_0023.ENC_Status_compact.Status/Counter_underflow <-> ENC Status compact/Status/Counter underflow
//     PlcTask Inputs/GVL_iXlinker.EtherCAT_Master_EPPxxxx.Beckhoff_EPP7xxx.Beckhoff_EPP7xxxEK1122.A_0007_EPP7041_3002_0023.ENC_Status_compact.Status/Counter_overflow <-> ENC Status compact/Status/Counter overflow
//     PlcTask Inputs/GVL_iXlinker.EtherCAT_Master_EPPxxxx.Beckhoff_EPP7xxx.Beckhoff_EPP7xxxEK1122.A_0007_EPP7041_3002_0023.ENC_Status_compact.Status/Extrapolation_stall <-> ENC Status compact/Status/Extrapolation stall
//     PlcTask Inputs/GVL_iXlinker.EtherCAT_Master_EPPxxxx.Beckhoff_EPP7xxx.Beckhoff_EPP7xxxEK1122.A_0007_EPP7041_3002_0023.ENC_Status_compact.Status/Status_of_input_A <-> ENC Status compact/Status/Status of input A
//     PlcTask Inputs/GVL_iXlinker.EtherCAT_Master_EPPxxxx.Beckhoff_EPP7xxx.Beckhoff_EPP7xxxEK1122.A_0007_EPP7041_3002_0023.ENC_Status_compact.Status/Status_of_input_B <-> ENC Status compact/Status/Status of input B
//     PlcTask Inputs/GVL_iXlinker.EtherCAT_Master_EPPxxxx.Beckhoff_EPP7xxx.Beckhoff_EPP7xxxEK1122.A_0007_EPP7041_3002_0023.ENC_Status_compact.Status/Status_of_input_C <-> ENC Status compact/Status/Status of input C
//     PlcTask Inputs/GVL_iXlinker.EtherCAT_Master_EPPxxxx.Beckhoff_EPP7xxx.Beckhoff_EPP7xxxEK1122.A_0007_EPP7041_3002_0023.ENC_Status_compact.Status/Status_of_extern_latch <-> ENC Status compact/Status/Status of extern latch
//     PlcTask Inputs/GVL_iXlinker.EtherCAT_Master_EPPxxxx.Beckhoff_EPP7xxx.Beckhoff_EPP7xxxEK1122.A_0007_EPP7041_3002_0023.ENC_Status_compact.Status/Sync_error <-> ENC Status compact/Status/Sync error
//     PlcTask Inputs/GVL_iXlinker.EtherCAT_Master_EPPxxxx.Beckhoff_EPP7xxx.Beckhoff_EPP7xxxEK1122.A_0007_EPP7041_3002_0023.ENC_Status_compact.Status/TxPDO_Toggle <-> ENC Status compact/Status/TxPDO Toggle
//     PlcTask Inputs/GVL_iXlinker.EtherCAT_Master_EPPxxxx.Beckhoff_EPP7xxx.Beckhoff_EPP7xxxEK1122.A_0007_EPP7041_3002_0023.ENC_Status_compact.Counter_value <-> ENC Status compact/Counter value
//     PlcTask Inputs/GVL_iXlinker.EtherCAT_Master_EPPxxxx.Beckhoff_EPP7xxx.Beckhoff_EPP7xxxEK1122.A_0007_EPP7041_3002_0023.ENC_Status_compact.Latch_value <-> ENC Status compact/Latch value
//     PlcTask Inputs/GVL_iXlinker.EtherCAT_Master_EPPxxxx.Beckhoff_EPP7xxx.Beckhoff_EPP7xxxEK1122.A_0007_EPP7041_3002_0023.STM_Status.Status/Ready_to_enable <-> STM Status/Status/Ready to enable
//     PlcTask Inputs/GVL_iXlinker.EtherCAT_Master_EPPxxxx.Beckhoff_EPP7xxx.Beckhoff_EPP7xxxEK1122.A_0007_EPP7041_3002_0023.STM_Status.Status/Ready <-> STM Status/Status/Ready
//     PlcTask Inputs/GVL_iXlinker.EtherCAT_Master_EPPxxxx.Beckhoff_EPP7xxx.Beckhoff_EPP7xxxEK1122.A_0007_EPP7041_3002_0023.STM_Status.Status/Warning <-> STM Status/Status/Warning
//     PlcTask Inputs/GVL_iXlinker.EtherCAT_Master_EPPxxxx.Beckhoff_EPP7xxx.Beckhoff_EPP7xxxEK1122.A_0007_EPP7041_3002_0023.STM_Status.Status/Error <-> STM Status/Status/Error
//     PlcTask Inputs/GVL_iXlinker.EtherCAT_Master_EPPxxxx.Beckhoff_EPP7xxx.Beckhoff_EPP7xxxEK1122.A_0007_EPP7041_3002_0023.STM_Status.Status/Moving_positive <-> STM Status/Status/Moving positive
//     PlcTask Inputs/GVL_iXlinker.EtherCAT_Master_EPPxxxx.Beckhoff_EPP7xxx.Beckhoff_EPP7xxxEK1122.A_0007_EPP7041_3002_0023.STM_Status.Status/Moving_negative <-> STM Status/Status/Moving negative
//     PlcTask Inputs/GVL_iXlinker.EtherCAT_Master_EPPxxxx.Beckhoff_EPP7xxx.Beckhoff_EPP7xxxEK1122.A_0007_EPP7041_3002_0023.STM_Status.Status/Torque_reduced <-> STM Status/Status/Torque reduced
//     PlcTask Inputs/GVL_iXlinker.EtherCAT_Master_EPPxxxx.Beckhoff_EPP7xxx.Beckhoff_EPP7xxxEK1122.A_0007_EPP7041_3002_0023.STM_Status.Status/Motor_stall <-> STM Status/Status/Motor stall
//     PlcTask Inputs/GVL_iXlinker.EtherCAT_Master_EPPxxxx.Beckhoff_EPP7xxx.Beckhoff_EPP7xxxEK1122.A_0007_EPP7041_3002_0023.STM_Status.Status/Digital_input_1 <-> STM Status/Status/Digital input 1
//     PlcTask Inputs/GVL_iXlinker.EtherCAT_Master_EPPxxxx.Beckhoff_EPP7xxx.Beckhoff_EPP7xxxEK1122.A_0007_EPP7041_3002_0023.STM_Status.Status/Digital_input_2 <-> STM Status/Status/Digital input 2
//     PlcTask Inputs/GVL_iXlinker.EtherCAT_Master_EPPxxxx.Beckhoff_EPP7xxx.Beckhoff_EPP7xxxEK1122.A_0007_EPP7041_3002_0023.STM_Status.Status/Sync_error <-> STM Status/Status/Sync error
//     PlcTask Inputs/GVL_iXlinker.EtherCAT_Master_EPPxxxx.Beckhoff_EPP7xxx.Beckhoff_EPP7xxxEK1122.A_0007_EPP7041_3002_0023.STM_Status.Status/TxPDO_Toggle <-> STM Status/Status/TxPDO Toggle
//     PlcTask Outputs/GVL_iXlinker.EtherCAT_Master_EPPxxxx.Beckhoff_EPP7xxx.Beckhoff_EPP7xxxEK1122.A_0007_EPP7041_3002_0023.ENC_Control_compact.Control/Enable_latch_C <-> ENC Control compact/Control/Enable latch C
//     PlcTask Outputs/GVL_iXlinker.EtherCAT_Master_EPPxxxx.Beckhoff_EPP7xxx.Beckhoff_EPP7xxxEK1122.A_0007_EPP7041_3002_0023.ENC_Control_compact.Control/Enable_latch_extern_on_positive_edge <-> ENC Control compact/Control/Enable latch extern on positive edge
//     PlcTask Outputs/GVL_iXlinker.EtherCAT_Master_EPPxxxx.Beckhoff_EPP7xxx.Beckhoff_EPP7xxxEK1122.A_0007_EPP7041_3002_0023.ENC_Control_compact.Control/Set_counter <-> ENC Control compact/Control/Set counter
//     PlcTask Outputs/GVL_iXlinker.EtherCAT_Master_EPPxxxx.Beckhoff_EPP7xxx.Beckhoff_EPP7xxxEK1122.A_0007_EPP7041_3002_0023.ENC_Control_compact.Control/Enable_latch_extern_on_negative_edge <-> ENC Control compact/Control/Enable latch extern on negative edge
//     PlcTask Outputs/GVL_iXlinker.EtherCAT_Master_EPPxxxx.Beckhoff_EPP7xxx.Beckhoff_EPP7xxxEK1122.A_0007_EPP7041_3002_0023.ENC_Control_compact.Set_counter_value <-> ENC Control compact/Set counter value
//     PlcTask Outputs/GVL_iXlinker.EtherCAT_Master_EPPxxxx.Beckhoff_EPP7xxx.Beckhoff_EPP7xxxEK1122.A_0007_EPP7041_3002_0023.STM_Control.Control/Enable <-> STM Control/Control/Enable
//     PlcTask Outputs/GVL_iXlinker.EtherCAT_Master_EPPxxxx.Beckhoff_EPP7xxx.Beckhoff_EPP7xxxEK1122.A_0007_EPP7041_3002_0023.STM_Control.Control/Reset <-> STM Control/Control/Reset
//     PlcTask Outputs/GVL_iXlinker.EtherCAT_Master_EPPxxxx.Beckhoff_EPP7xxx.Beckhoff_EPP7xxxEK1122.A_0007_EPP7041_3002_0023.STM_Control.Control/Reduce_torque <-> STM Control/Control/Reduce torque
//     PlcTask Outputs/GVL_iXlinker.EtherCAT_Master_EPPxxxx.Beckhoff_EPP7xxx.Beckhoff_EPP7xxxEK1122.A_0007_EPP7041_3002_0023.STM_Control.Control/Digital_output_1 <-> STM Control/Control/Digital output 1
//     PlcTask Outputs/GVL_iXlinker.EtherCAT_Master_EPPxxxx.Beckhoff_EPP7xxx.Beckhoff_EPP7xxxEK1122.A_0007_EPP7041_3002_0023.STM_Velocity.Velocity <-> STM Velocity/Velocity
//     PlcTask Inputs/GVL_iXlinker.EtherCAT_Master_EPPxxxx.Beckhoff_EPP7xxx.Beckhoff_EPP7xxxEK1122.A_0007_EPP7041_3002_0023.WcState.WcState <-> WcState/WcState
//     PlcTask Inputs/GVL_iXlinker.EtherCAT_Master_EPPxxxx.Beckhoff_EPP7xxx.Beckhoff_EPP7xxxEK1122.A_0007_EPP7041_3002_0023.WcState.InputToggle <-> WcState/InputToggle
//     PlcTask Inputs/GVL_iXlinker.EtherCAT_Master_EPPxxxx.Beckhoff_EPP7xxx.Beckhoff_EPP7xxxEK1122.A_0007_EPP7041_3002_0023.InfoData.AdsAddr <-> InfoData/AdsAddr
//     PlcTask Inputs/GVL_iXlinker.EtherCAT_Master_EPPxxxx.Beckhoff_EPP7xxx.Beckhoff_EPP7xxxEK1122.A_0007_EPP7041_3002_0023.InfoData.Chn0 <-> InfoData/Chn0
//     PlcTask Inputs/GVL_iXlinker.EtherCAT_Master_EPPxxxx.Beckhoff_EPP7xxx.Beckhoff_EPP7xxxEK1122.A_0007_EPP7041_3002_0023.InfoData.Chn1 <-> InfoData/Chn1
//     PlcTask Inputs/GVL_iXlinker.EtherCAT_Master_EPPxxxx.Beckhoff_EPP7xxx.Beckhoff_EPP7xxxEK1122.A_0007_EPP7041_3002_0023.InfoData.State <-> InfoData/State
//   PLC/PLC Instance <-> EtherCAT Master EPPxxxx/Beckhoff EPP7xxx/Beckhoff EPP7xxxEK1122/A_0008(EPP7342-0002-0016)
//     PlcTask Inputs/GVL_iXlinker.EtherCAT_Master_EPPxxxx.Beckhoff_EPP7xxx.Beckhoff_EPP7xxxEK1122.A_0008_EPP7342_0002_0016.ENC_Status_compact_Channel_1.Status/Latch_extern_valid <-> ENC Status compact Channel 1/Status/Latch extern valid
//     PlcTask Inputs/GVL_iXlinker.EtherCAT_Master_EPPxxxx.Beckhoff_EPP7xxx.Beckhoff_EPP7xxxEK1122.A_0008_EPP7342_0002_0016.ENC_Status_compact_Channel_2.Status/Latch_extern_valid <-> ENC Status compact Channel 2/Status/Latch extern valid
//     PlcTask Inputs/GVL_iXlinker.EtherCAT_Master_EPPxxxx.Beckhoff_EPP7xxx.Beckhoff_EPP7xxxEK1122.A_0008_EPP7342_0002_0016.ENC_Status_compact_Channel_1.Status/Set_counter_done <-> ENC Status compact Channel 1/Status/Set counter done
//     PlcTask Inputs/GVL_iXlinker.EtherCAT_Master_EPPxxxx.Beckhoff_EPP7xxx.Beckhoff_EPP7xxxEK1122.A_0008_EPP7342_0002_0016.ENC_Status_compact_Channel_2.Status/Set_counter_done <-> ENC Status compact Channel 2/Status/Set counter done
//     PlcTask Inputs/GVL_iXlinker.EtherCAT_Master_EPPxxxx.Beckhoff_EPP7xxx.Beckhoff_EPP7xxxEK1122.A_0008_EPP7342_0002_0016.ENC_Status_compact_Channel_1.Status/Counter_underflow <-> ENC Status compact Channel 1/Status/Counter underflow
//     PlcTask Inputs/GVL_iXlinker.EtherCAT_Master_EPPxxxx.Beckhoff_EPP7xxx.Beckhoff_EPP7xxxEK1122.A_0008_EPP7342_0002_0016.ENC_Status_compact_Channel_2.Status/Counter_underflow <-> ENC Status compact Channel 2/Status/Counter underflow
//     PlcTask Inputs/GVL_iXlinker.EtherCAT_Master_EPPxxxx.Beckhoff_EPP7xxx.Beckhoff_EPP7xxxEK1122.A_0008_EPP7342_0002_0016.ENC_Status_compact_Channel_1.Status/Counter_overflow <-> ENC Status compact Channel 1/Status/Counter overflow
//     PlcTask Inputs/GVL_iXlinker.EtherCAT_Master_EPPxxxx.Beckhoff_EPP7xxx.Beckhoff_EPP7xxxEK1122.A_0008_EPP7342_0002_0016.ENC_Status_compact_Channel_2.Status/Counter_overflow <-> ENC Status compact Channel 2/Status/Counter overflow
//     PlcTask Inputs/GVL_iXlinker.EtherCAT_Master_EPPxxxx.Beckhoff_EPP7xxx.Beckhoff_EPP7xxxEK1122.A_0008_EPP7342_0002_0016.ENC_Status_compact_Channel_1.Status/Extrapolation_stall <-> ENC Status compact Channel 1/Status/Extrapolation stall
//     PlcTask Inputs/GVL_iXlinker.EtherCAT_Master_EPPxxxx.Beckhoff_EPP7xxx.Beckhoff_EPP7xxxEK1122.A_0008_EPP7342_0002_0016.ENC_Status_compact_Channel_2.Status/Extrapolation_stall <-> ENC Status compact Channel 2/Status/Extrapolation stall
//     PlcTask Inputs/GVL_iXlinker.EtherCAT_Master_EPPxxxx.Beckhoff_EPP7xxx.Beckhoff_EPP7xxxEK1122.A_0008_EPP7342_0002_0016.ENC_Status_compact_Channel_1.Status/Status_of_input_A <-> ENC Status compact Channel 1/Status/Status of input A
//     PlcTask Inputs/GVL_iXlinker.EtherCAT_Master_EPPxxxx.Beckhoff_EPP7xxx.Beckhoff_EPP7xxxEK1122.A_0008_EPP7342_0002_0016.ENC_Status_compact_Channel_2.Status/Status_of_input_A <-> ENC Status compact Channel 2/Status/Status of input A
//     PlcTask Inputs/GVL_iXlinker.EtherCAT_Master_EPPxxxx.Beckhoff_EPP7xxx.Beckhoff_EPP7xxxEK1122.A_0008_EPP7342_0002_0016.ENC_Status_compact_Channel_1.Status/Status_of_input_B <-> ENC Status compact Channel 1/Status/Status of input B
//     PlcTask Inputs/GVL_iXlinker.EtherCAT_Master_EPPxxxx.Beckhoff_EPP7xxx.Beckhoff_EPP7xxxEK1122.A_0008_EPP7342_0002_0016.ENC_Status_compact_Channel_2.Status/Status_of_input_B <-> ENC Status compact Channel 2/Status/Status of input B
//     PlcTask Inputs/GVL_iXlinker.EtherCAT_Master_EPPxxxx.Beckhoff_EPP7xxx.Beckhoff_EPP7xxxEK1122.A_0008_EPP7342_0002_0016.ENC_Status_compact_Channel_1.Status/Status_of_extern_latch <-> ENC Status compact Channel 1/Status/Status of extern latch
//     PlcTask Inputs/GVL_iXlinker.EtherCAT_Master_EPPxxxx.Beckhoff_EPP7xxx.Beckhoff_EPP7xxxEK1122.A_0008_EPP7342_0002_0016.ENC_Status_compact_Channel_2.Status/Status_of_extern_latch <-> ENC Status compact Channel 2/Status/Status of extern latch
//     PlcTask Inputs/GVL_iXlinker.EtherCAT_Master_EPPxxxx.Beckhoff_EPP7xxx.Beckhoff_EPP7xxxEK1122.A_0008_EPP7342_0002_0016.ENC_Status_compact_Channel_1.Status/Sync_error <-> ENC Status compact Channel 1/Status/Sync error
//     PlcTask Inputs/GVL_iXlinker.EtherCAT_Master_EPPxxxx.Beckhoff_EPP7xxx.Beckhoff_EPP7xxxEK1122.A_0008_EPP7342_0002_0016.ENC_Status_compact_Channel_2.Status/Sync_error <-> ENC Status compact Channel 2/Status/Sync error
//     PlcTask Inputs/GVL_iXlinker.EtherCAT_Master_EPPxxxx.Beckhoff_EPP7xxx.Beckhoff_EPP7xxxEK1122.A_0008_EPP7342_0002_0016.ENC_Status_compact_Channel_1.Status/TxPDO_Toggle <-> ENC Status compact Channel 1/Status/TxPDO Toggle
//     PlcTask Inputs/GVL_iXlinker.EtherCAT_Master_EPPxxxx.Beckhoff_EPP7xxx.Beckhoff_EPP7xxxEK1122.A_0008_EPP7342_0002_0016.ENC_Status_compact_Channel_2.Status/TxPDO_Toggle <-> ENC Status compact Channel 2/Status/TxPDO Toggle
//     PlcTask Inputs/GVL_iXlinker.EtherCAT_Master_EPPxxxx.Beckhoff_EPP7xxx.Beckhoff_EPP7xxxEK1122.A_0008_EPP7342_0002_0016.ENC_Status_compact_Channel_1.Counter_value <-> ENC Status compact Channel 1/Counter value
//     PlcTask Inputs/GVL_iXlinker.EtherCAT_Master_EPPxxxx.Beckhoff_EPP7xxx.Beckhoff_EPP7xxxEK1122.A_0008_EPP7342_0002_0016.ENC_Status_compact_Channel_2.Counter_value <-> ENC Status compact Channel 2/Counter value
//     PlcTask Inputs/GVL_iXlinker.EtherCAT_Master_EPPxxxx.Beckhoff_EPP7xxx.Beckhoff_EPP7xxxEK1122.A_0008_EPP7342_0002_0016.ENC_Status_compact_Channel_1.Latch_value <-> ENC Status compact Channel 1/Latch value
//     PlcTask Inputs/GVL_iXlinker.EtherCAT_Master_EPPxxxx.Beckhoff_EPP7xxx.Beckhoff_EPP7xxxEK1122.A_0008_EPP7342_0002_0016.ENC_Status_compact_Channel_2.Latch_value <-> ENC Status compact Channel 2/Latch value
//     PlcTask Inputs/GVL_iXlinker.EtherCAT_Master_EPPxxxx.Beckhoff_EPP7xxx.Beckhoff_EPP7xxxEK1122.A_0008_EPP7342_0002_0016.DCM_Status_Channel_1.Status/Ready_to_enable <-> DCM Status Channel 1/Status/Ready to enable
//     PlcTask Inputs/GVL_iXlinker.EtherCAT_Master_EPPxxxx.Beckhoff_EPP7xxx.Beckhoff_EPP7xxxEK1122.A_0008_EPP7342_0002_0016.DCM_Status_Channel_2.Status/Ready_to_enable <-> DCM Status Channel 2/Status/Ready to enable
//     PlcTask Inputs/GVL_iXlinker.EtherCAT_Master_EPPxxxx.Beckhoff_EPP7xxx.Beckhoff_EPP7xxxEK1122.A_0008_EPP7342_0002_0016.DCM_Status_Channel_1.Status/Ready <-> DCM Status Channel 1/Status/Ready
//     PlcTask Inputs/GVL_iXlinker.EtherCAT_Master_EPPxxxx.Beckhoff_EPP7xxx.Beckhoff_EPP7xxxEK1122.A_0008_EPP7342_0002_0016.DCM_Status_Channel_2.Status/Ready <-> DCM Status Channel 2/Status/Ready
//     PlcTask Inputs/GVL_iXlinker.EtherCAT_Master_EPPxxxx.Beckhoff_EPP7xxx.Beckhoff_EPP7xxxEK1122.A_0008_EPP7342_0002_0016.DCM_Status_Channel_1.Status/Warning <-> DCM Status Channel 1/Status/Warning
//     PlcTask Inputs/GVL_iXlinker.EtherCAT_Master_EPPxxxx.Beckhoff_EPP7xxx.Beckhoff_EPP7xxxEK1122.A_0008_EPP7342_0002_0016.DCM_Status_Channel_2.Status/Warning <-> DCM Status Channel 2/Status/Warning
//     PlcTask Inputs/GVL_iXlinker.EtherCAT_Master_EPPxxxx.Beckhoff_EPP7xxx.Beckhoff_EPP7xxxEK1122.A_0008_EPP7342_0002_0016.DCM_Status_Channel_1.Status/Error <-> DCM Status Channel 1/Status/Error
//     PlcTask Inputs/GVL_iXlinker.EtherCAT_Master_EPPxxxx.Beckhoff_EPP7xxx.Beckhoff_EPP7xxxEK1122.A_0008_EPP7342_0002_0016.DCM_Status_Channel_2.Status/Error <-> DCM Status Channel 2/Status/Error
//     PlcTask Inputs/GVL_iXlinker.EtherCAT_Master_EPPxxxx.Beckhoff_EPP7xxx.Beckhoff_EPP7xxxEK1122.A_0008_EPP7342_0002_0016.DCM_Status_Channel_1.Status/Moving_positive <-> DCM Status Channel 1/Status/Moving positive
//     PlcTask Inputs/GVL_iXlinker.EtherCAT_Master_EPPxxxx.Beckhoff_EPP7xxx.Beckhoff_EPP7xxxEK1122.A_0008_EPP7342_0002_0016.DCM_Status_Channel_2.Status/Moving_positive <-> DCM Status Channel 2/Status/Moving positive
//     PlcTask Inputs/GVL_iXlinker.EtherCAT_Master_EPPxxxx.Beckhoff_EPP7xxx.Beckhoff_EPP7xxxEK1122.A_0008_EPP7342_0002_0016.DCM_Status_Channel_1.Status/Moving_negative <-> DCM Status Channel 1/Status/Moving negative
//     PlcTask Inputs/GVL_iXlinker.EtherCAT_Master_EPPxxxx.Beckhoff_EPP7xxx.Beckhoff_EPP7xxxEK1122.A_0008_EPP7342_0002_0016.DCM_Status_Channel_2.Status/Moving_negative <-> DCM Status Channel 2/Status/Moving negative
//     PlcTask Inputs/GVL_iXlinker.EtherCAT_Master_EPPxxxx.Beckhoff_EPP7xxx.Beckhoff_EPP7xxxEK1122.A_0008_EPP7342_0002_0016.DCM_Status_Channel_1.Status/Torque_reduced <-> DCM Status Channel 1/Status/Torque reduced
//     PlcTask Inputs/GVL_iXlinker.EtherCAT_Master_EPPxxxx.Beckhoff_EPP7xxx.Beckhoff_EPP7xxxEK1122.A_0008_EPP7342_0002_0016.DCM_Status_Channel_2.Status/Torque_reduced <-> DCM Status Channel 2/Status/Torque reduced
//     PlcTask Inputs/GVL_iXlinker.EtherCAT_Master_EPPxxxx.Beckhoff_EPP7xxx.Beckhoff_EPP7xxxEK1122.A_0008_EPP7342_0002_0016.DCM_Status_Channel_1.Status/Digital_input_1 <-> DCM Status Channel 1/Status/Digital input 1
//     PlcTask Inputs/GVL_iXlinker.EtherCAT_Master_EPPxxxx.Beckhoff_EPP7xxx.Beckhoff_EPP7xxxEK1122.A_0008_EPP7342_0002_0016.DCM_Status_Channel_1.Status/Digital_input_2 <-> DCM Status Channel 1/Status/Digital input 2
//     PlcTask Inputs/GVL_iXlinker.EtherCAT_Master_EPPxxxx.Beckhoff_EPP7xxx.Beckhoff_EPP7xxxEK1122.A_0008_EPP7342_0002_0016.DCM_Status_Channel_2.Status/Digital_input_1 <-> DCM Status Channel 2/Status/Digital input 1
//     PlcTask Inputs/GVL_iXlinker.EtherCAT_Master_EPPxxxx.Beckhoff_EPP7xxx.Beckhoff_EPP7xxxEK1122.A_0008_EPP7342_0002_0016.DCM_Status_Channel_2.Status/Digital_input_2 <-> DCM Status Channel 2/Status/Digital input 2
//     PlcTask Inputs/GVL_iXlinker.EtherCAT_Master_EPPxxxx.Beckhoff_EPP7xxx.Beckhoff_EPP7xxxEK1122.A_0008_EPP7342_0002_0016.DCM_Status_Channel_1.Status/Sync_error <-> DCM Status Channel 1/Status/Sync error
//     PlcTask Inputs/GVL_iXlinker.EtherCAT_Master_EPPxxxx.Beckhoff_EPP7xxx.Beckhoff_EPP7xxxEK1122.A_0008_EPP7342_0002_0016.DCM_Status_Channel_2.Status/Sync_error <-> DCM Status Channel 2/Status/Sync error
//     PlcTask Inputs/GVL_iXlinker.EtherCAT_Master_EPPxxxx.Beckhoff_EPP7xxx.Beckhoff_EPP7xxxEK1122.A_0008_EPP7342_0002_0016.DCM_Status_Channel_1.Status/TxPDO_Toggle <-> DCM Status Channel 1/Status/TxPDO Toggle
//     PlcTask Inputs/GVL_iXlinker.EtherCAT_Master_EPPxxxx.Beckhoff_EPP7xxx.Beckhoff_EPP7xxxEK1122.A_0008_EPP7342_0002_0016.DCM_Status_Channel_2.Status/TxPDO_Toggle <-> DCM Status Channel 2/Status/TxPDO Toggle
//     PlcTask Outputs/GVL_iXlinker.EtherCAT_Master_EPPxxxx.Beckhoff_EPP7xxx.Beckhoff_EPP7xxxEK1122.A_0008_EPP7342_0002_0016.ENC_Control_compact_Channel_1.Control/Enable_latch_extern_on_positive_edge <-> ENC Control compact Channel 1/Control/Enable latch extern on positive edge
//     PlcTask Outputs/GVL_iXlinker.EtherCAT_Master_EPPxxxx.Beckhoff_EPP7xxx.Beckhoff_EPP7xxxEK1122.A_0008_EPP7342_0002_0016.ENC_Control_compact_Channel_2.Control/Enable_latch_extern_on_positive_edge <-> ENC Control compact Channel 2/Control/Enable latch extern on positive edge
//     PlcTask Outputs/GVL_iXlinker.EtherCAT_Master_EPPxxxx.Beckhoff_EPP7xxx.Beckhoff_EPP7xxxEK1122.A_0008_EPP7342_0002_0016.ENC_Control_compact_Channel_1.Control/Set_counter <-> ENC Control compact Channel 1/Control/Set counter
//     PlcTask Outputs/GVL_iXlinker.EtherCAT_Master_EPPxxxx.Beckhoff_EPP7xxx.Beckhoff_EPP7xxxEK1122.A_0008_EPP7342_0002_0016.ENC_Control_compact_Channel_2.Control/Set_counter <-> ENC Control compact Channel 2/Control/Set counter
//     PlcTask Outputs/GVL_iXlinker.EtherCAT_Master_EPPxxxx.Beckhoff_EPP7xxx.Beckhoff_EPP7xxxEK1122.A_0008_EPP7342_0002_0016.ENC_Control_compact_Channel_1.Control/Enable_latch_extern_on_negative_edge <-> ENC Control compact Channel 1/Control/Enable latch extern on negative edge
//     PlcTask Outputs/GVL_iXlinker.EtherCAT_Master_EPPxxxx.Beckhoff_EPP7xxx.Beckhoff_EPP7xxxEK1122.A_0008_EPP7342_0002_0016.ENC_Control_compact_Channel_2.Control/Enable_latch_extern_on_negative_edge <-> ENC Control compact Channel 2/Control/Enable latch extern on negative edge
//     PlcTask Outputs/GVL_iXlinker.EtherCAT_Master_EPPxxxx.Beckhoff_EPP7xxx.Beckhoff_EPP7xxxEK1122.A_0008_EPP7342_0002_0016.ENC_Control_compact_Channel_1.Set_counter_value <-> ENC Control compact Channel 1/Set counter value
//     PlcTask Outputs/GVL_iXlinker.EtherCAT_Master_EPPxxxx.Beckhoff_EPP7xxx.Beckhoff_EPP7xxxEK1122.A_0008_EPP7342_0002_0016.ENC_Control_compact_Channel_2.Set_counter_value <-> ENC Control compact Channel 2/Set counter value
//     PlcTask Outputs/GVL_iXlinker.EtherCAT_Master_EPPxxxx.Beckhoff_EPP7xxx.Beckhoff_EPP7xxxEK1122.A_0008_EPP7342_0002_0016.DCM_Control_Channel_1.Control/Enable <-> DCM Control Channel 1/Control/Enable
//     PlcTask Outputs/GVL_iXlinker.EtherCAT_Master_EPPxxxx.Beckhoff_EPP7xxx.Beckhoff_EPP7xxxEK1122.A_0008_EPP7342_0002_0016.DCM_Control_Channel_2.Control/Enable <-> DCM Control Channel 2/Control/Enable
//     PlcTask Outputs/GVL_iXlinker.EtherCAT_Master_EPPxxxx.Beckhoff_EPP7xxx.Beckhoff_EPP7xxxEK1122.A_0008_EPP7342_0002_0016.DCM_Control_Channel_1.Control/Reset <-> DCM Control Channel 1/Control/Reset
//     PlcTask Outputs/GVL_iXlinker.EtherCAT_Master_EPPxxxx.Beckhoff_EPP7xxx.Beckhoff_EPP7xxxEK1122.A_0008_EPP7342_0002_0016.DCM_Control_Channel_2.Control/Reset <-> DCM Control Channel 2/Control/Reset
//     PlcTask Outputs/GVL_iXlinker.EtherCAT_Master_EPPxxxx.Beckhoff_EPP7xxx.Beckhoff_EPP7xxxEK1122.A_0008_EPP7342_0002_0016.DCM_Control_Channel_1.Control/Reduce_torque <-> DCM Control Channel 1/Control/Reduce torque
//     PlcTask Outputs/GVL_iXlinker.EtherCAT_Master_EPPxxxx.Beckhoff_EPP7xxx.Beckhoff_EPP7xxxEK1122.A_0008_EPP7342_0002_0016.DCM_Control_Channel_2.Control/Reduce_torque <-> DCM Control Channel 2/Control/Reduce torque
//     PlcTask Outputs/GVL_iXlinker.EtherCAT_Master_EPPxxxx.Beckhoff_EPP7xxx.Beckhoff_EPP7xxxEK1122.A_0008_EPP7342_0002_0016.DCM_Velocity_Channel_1.Velocity <-> DCM Velocity Channel 1/Velocity
//     PlcTask Outputs/GVL_iXlinker.EtherCAT_Master_EPPxxxx.Beckhoff_EPP7xxx.Beckhoff_EPP7xxxEK1122.A_0008_EPP7342_0002_0016.DCM_Velocity_Channel_2.Velocity <-> DCM Velocity Channel 2/Velocity
//     PlcTask Inputs/GVL_iXlinker.EtherCAT_Master_EPPxxxx.Beckhoff_EPP7xxx.Beckhoff_EPP7xxxEK1122.A_0008_EPP7342_0002_0016.WcState.WcState <-> WcState/WcState
//     PlcTask Inputs/GVL_iXlinker.EtherCAT_Master_EPPxxxx.Beckhoff_EPP7xxx.Beckhoff_EPP7xxxEK1122.A_0008_EPP7342_0002_0016.WcState.InputToggle <-> WcState/InputToggle
//     PlcTask Inputs/GVL_iXlinker.EtherCAT_Master_EPPxxxx.Beckhoff_EPP7xxx.Beckhoff_EPP7xxxEK1122.A_0008_EPP7342_0002_0016.InfoData.AdsAddr <-> InfoData/AdsAddr
//     PlcTask Inputs/GVL_iXlinker.EtherCAT_Master_EPPxxxx.Beckhoff_EPP7xxx.Beckhoff_EPP7xxxEK1122.A_0008_EPP7342_0002_0016.InfoData.Chn0 <-> InfoData/Chn0
//     PlcTask Inputs/GVL_iXlinker.EtherCAT_Master_EPPxxxx.Beckhoff_EPP7xxx.Beckhoff_EPP7xxxEK1122.A_0008_EPP7342_0002_0016.InfoData.Chn1 <-> InfoData/Chn1
//     PlcTask Inputs/GVL_iXlinker.EtherCAT_Master_EPPxxxx.Beckhoff_EPP7xxx.Beckhoff_EPP7xxxEK1122.A_0008_EPP7342_0002_0016.InfoData.Chn2 <-> InfoData/Chn2
//     PlcTask Inputs/GVL_iXlinker.EtherCAT_Master_EPPxxxx.Beckhoff_EPP7xxx.Beckhoff_EPP7xxxEK1122.A_0008_EPP7342_0002_0016.InfoData.Chn3 <-> InfoData/Chn3
//     PlcTask Inputs/GVL_iXlinker.EtherCAT_Master_EPPxxxx.Beckhoff_EPP7xxx.Beckhoff_EPP7xxxEK1122.A_0008_EPP7342_0002_0016.InfoData.State <-> InfoData/State
//   PLC/PLC Instance <-> EtherCAT Master EPPxxxx/Beckhoff EPP7xxx/Beckhoff EPP7xxxEK1122/A_0009(EPP7342-0002-0017)
//     PlcTask Inputs/GVL_iXlinker.EtherCAT_Master_EPPxxxx.Beckhoff_EPP7xxx.Beckhoff_EPP7xxxEK1122.A_0009_EPP7342_0002_0017.ENC_Status_compact_Channel_1.Status/Latch_extern_valid <-> ENC Status compact Channel 1/Status/Latch extern valid
//     PlcTask Inputs/GVL_iXlinker.EtherCAT_Master_EPPxxxx.Beckhoff_EPP7xxx.Beckhoff_EPP7xxxEK1122.A_0009_EPP7342_0002_0017.ENC_Status_compact_Channel_2.Status/Latch_extern_valid <-> ENC Status compact Channel 2/Status/Latch extern valid
//     PlcTask Inputs/GVL_iXlinker.EtherCAT_Master_EPPxxxx.Beckhoff_EPP7xxx.Beckhoff_EPP7xxxEK1122.A_0009_EPP7342_0002_0017.ENC_Status_compact_Channel_1.Status/Set_counter_done <-> ENC Status compact Channel 1/Status/Set counter done
//     PlcTask Inputs/GVL_iXlinker.EtherCAT_Master_EPPxxxx.Beckhoff_EPP7xxx.Beckhoff_EPP7xxxEK1122.A_0009_EPP7342_0002_0017.ENC_Status_compact_Channel_2.Status/Set_counter_done <-> ENC Status compact Channel 2/Status/Set counter done
//     PlcTask Inputs/GVL_iXlinker.EtherCAT_Master_EPPxxxx.Beckhoff_EPP7xxx.Beckhoff_EPP7xxxEK1122.A_0009_EPP7342_0002_0017.ENC_Status_compact_Channel_1.Status/Counter_underflow <-> ENC Status compact Channel 1/Status/Counter underflow
//     PlcTask Inputs/GVL_iXlinker.EtherCAT_Master_EPPxxxx.Beckhoff_EPP7xxx.Beckhoff_EPP7xxxEK1122.A_0009_EPP7342_0002_0017.ENC_Status_compact_Channel_2.Status/Counter_underflow <-> ENC Status compact Channel 2/Status/Counter underflow
//     PlcTask Inputs/GVL_iXlinker.EtherCAT_Master_EPPxxxx.Beckhoff_EPP7xxx.Beckhoff_EPP7xxxEK1122.A_0009_EPP7342_0002_0017.ENC_Status_compact_Channel_1.Status/Counter_overflow <-> ENC Status compact Channel 1/Status/Counter overflow
//     PlcTask Inputs/GVL_iXlinker.EtherCAT_Master_EPPxxxx.Beckhoff_EPP7xxx.Beckhoff_EPP7xxxEK1122.A_0009_EPP7342_0002_0017.ENC_Status_compact_Channel_2.Status/Counter_overflow <-> ENC Status compact Channel 2/Status/Counter overflow
//     PlcTask Inputs/GVL_iXlinker.EtherCAT_Master_EPPxxxx.Beckhoff_EPP7xxx.Beckhoff_EPP7xxxEK1122.A_0009_EPP7342_0002_0017.ENC_Status_compact_Channel_1.Status/Extrapolation_stall <-> ENC Status compact Channel 1/Status/Extrapolation stall
//     PlcTask Inputs/GVL_iXlinker.EtherCAT_Master_EPPxxxx.Beckhoff_EPP7xxx.Beckhoff_EPP7xxxEK1122.A_0009_EPP7342_0002_0017.ENC_Status_compact_Channel_2.Status/Extrapolation_stall <-> ENC Status compact Channel 2/Status/Extrapolation stall
//     PlcTask Inputs/GVL_iXlinker.EtherCAT_Master_EPPxxxx.Beckhoff_EPP7xxx.Beckhoff_EPP7xxxEK1122.A_0009_EPP7342_0002_0017.ENC_Status_compact_Channel_1.Status/Status_of_input_A <-> ENC Status compact Channel 1/Status/Status of input A
//     PlcTask Inputs/GVL_iXlinker.EtherCAT_Master_EPPxxxx.Beckhoff_EPP7xxx.Beckhoff_EPP7xxxEK1122.A_0009_EPP7342_0002_0017.ENC_Status_compact_Channel_2.Status/Status_of_input_A <-> ENC Status compact Channel 2/Status/Status of input A
//     PlcTask Inputs/GVL_iXlinker.EtherCAT_Master_EPPxxxx.Beckhoff_EPP7xxx.Beckhoff_EPP7xxxEK1122.A_0009_EPP7342_0002_0017.ENC_Status_compact_Channel_1.Status/Status_of_input_B <-> ENC Status compact Channel 1/Status/Status of input B
//     PlcTask Inputs/GVL_iXlinker.EtherCAT_Master_EPPxxxx.Beckhoff_EPP7xxx.Beckhoff_EPP7xxxEK1122.A_0009_EPP7342_0002_0017.ENC_Status_compact_Channel_2.Status/Status_of_input_B <-> ENC Status compact Channel 2/Status/Status of input B
//     PlcTask Inputs/GVL_iXlinker.EtherCAT_Master_EPPxxxx.Beckhoff_EPP7xxx.Beckhoff_EPP7xxxEK1122.A_0009_EPP7342_0002_0017.ENC_Status_compact_Channel_1.Status/Status_of_extern_latch <-> ENC Status compact Channel 1/Status/Status of extern latch
//     PlcTask Inputs/GVL_iXlinker.EtherCAT_Master_EPPxxxx.Beckhoff_EPP7xxx.Beckhoff_EPP7xxxEK1122.A_0009_EPP7342_0002_0017.ENC_Status_compact_Channel_2.Status/Status_of_extern_latch <-> ENC Status compact Channel 2/Status/Status of extern latch
//     PlcTask Inputs/GVL_iXlinker.EtherCAT_Master_EPPxxxx.Beckhoff_EPP7xxx.Beckhoff_EPP7xxxEK1122.A_0009_EPP7342_0002_0017.ENC_Status_compact_Channel_1.Status/Sync_error <-> ENC Status compact Channel 1/Status/Sync error
//     PlcTask Inputs/GVL_iXlinker.EtherCAT_Master_EPPxxxx.Beckhoff_EPP7xxx.Beckhoff_EPP7xxxEK1122.A_0009_EPP7342_0002_0017.ENC_Status_compact_Channel_2.Status/Sync_error <-> ENC Status compact Channel 2/Status/Sync error
//     PlcTask Inputs/GVL_iXlinker.EtherCAT_Master_EPPxxxx.Beckhoff_EPP7xxx.Beckhoff_EPP7xxxEK1122.A_0009_EPP7342_0002_0017.ENC_Status_compact_Channel_1.Status/TxPDO_Toggle <-> ENC Status compact Channel 1/Status/TxPDO Toggle
//     PlcTask Inputs/GVL_iXlinker.EtherCAT_Master_EPPxxxx.Beckhoff_EPP7xxx.Beckhoff_EPP7xxxEK1122.A_0009_EPP7342_0002_0017.ENC_Status_compact_Channel_2.Status/TxPDO_Toggle <-> ENC Status compact Channel 2/Status/TxPDO Toggle
//     PlcTask Inputs/GVL_iXlinker.EtherCAT_Master_EPPxxxx.Beckhoff_EPP7xxx.Beckhoff_EPP7xxxEK1122.A_0009_EPP7342_0002_0017.ENC_Status_compact_Channel_1.Counter_value <-> ENC Status compact Channel 1/Counter value
//     PlcTask Inputs/GVL_iXlinker.EtherCAT_Master_EPPxxxx.Beckhoff_EPP7xxx.Beckhoff_EPP7xxxEK1122.A_0009_EPP7342_0002_0017.ENC_Status_compact_Channel_2.Counter_value <-> ENC Status compact Channel 2/Counter value
//     PlcTask Inputs/GVL_iXlinker.EtherCAT_Master_EPPxxxx.Beckhoff_EPP7xxx.Beckhoff_EPP7xxxEK1122.A_0009_EPP7342_0002_0017.ENC_Status_compact_Channel_1.Latch_value <-> ENC Status compact Channel 1/Latch value
//     PlcTask Inputs/GVL_iXlinker.EtherCAT_Master_EPPxxxx.Beckhoff_EPP7xxx.Beckhoff_EPP7xxxEK1122.A_0009_EPP7342_0002_0017.ENC_Status_compact_Channel_2.Latch_value <-> ENC Status compact Channel 2/Latch value
//     PlcTask Inputs/GVL_iXlinker.EtherCAT_Master_EPPxxxx.Beckhoff_EPP7xxx.Beckhoff_EPP7xxxEK1122.A_0009_EPP7342_0002_0017.DCM_Status_Channel_1.Status/Ready_to_enable <-> DCM Status Channel 1/Status/Ready to enable
//     PlcTask Inputs/GVL_iXlinker.EtherCAT_Master_EPPxxxx.Beckhoff_EPP7xxx.Beckhoff_EPP7xxxEK1122.A_0009_EPP7342_0002_0017.DCM_Status_Channel_2.Status/Ready_to_enable <-> DCM Status Channel 2/Status/Ready to enable
//     PlcTask Inputs/GVL_iXlinker.EtherCAT_Master_EPPxxxx.Beckhoff_EPP7xxx.Beckhoff_EPP7xxxEK1122.A_0009_EPP7342_0002_0017.DCM_Status_Channel_1.Status/Ready <-> DCM Status Channel 1/Status/Ready
//     PlcTask Inputs/GVL_iXlinker.EtherCAT_Master_EPPxxxx.Beckhoff_EPP7xxx.Beckhoff_EPP7xxxEK1122.A_0009_EPP7342_0002_0017.DCM_Status_Channel_2.Status/Ready <-> DCM Status Channel 2/Status/Ready
//     PlcTask Inputs/GVL_iXlinker.EtherCAT_Master_EPPxxxx.Beckhoff_EPP7xxx.Beckhoff_EPP7xxxEK1122.A_0009_EPP7342_0002_0017.DCM_Status_Channel_1.Status/Warning <-> DCM Status Channel 1/Status/Warning
//     PlcTask Inputs/GVL_iXlinker.EtherCAT_Master_EPPxxxx.Beckhoff_EPP7xxx.Beckhoff_EPP7xxxEK1122.A_0009_EPP7342_0002_0017.DCM_Status_Channel_2.Status/Warning <-> DCM Status Channel 2/Status/Warning
//     PlcTask Inputs/GVL_iXlinker.EtherCAT_Master_EPPxxxx.Beckhoff_EPP7xxx.Beckhoff_EPP7xxxEK1122.A_0009_EPP7342_0002_0017.DCM_Status_Channel_1.Status/Error <-> DCM Status Channel 1/Status/Error
//     PlcTask Inputs/GVL_iXlinker.EtherCAT_Master_EPPxxxx.Beckhoff_EPP7xxx.Beckhoff_EPP7xxxEK1122.A_0009_EPP7342_0002_0017.DCM_Status_Channel_2.Status/Error <-> DCM Status Channel 2/Status/Error
//     PlcTask Inputs/GVL_iXlinker.EtherCAT_Master_EPPxxxx.Beckhoff_EPP7xxx.Beckhoff_EPP7xxxEK1122.A_0009_EPP7342_0002_0017.DCM_Status_Channel_1.Status/Moving_positive <-> DCM Status Channel 1/Status/Moving positive
//     PlcTask Inputs/GVL_iXlinker.EtherCAT_Master_EPPxxxx.Beckhoff_EPP7xxx.Beckhoff_EPP7xxxEK1122.A_0009_EPP7342_0002_0017.DCM_Status_Channel_2.Status/Moving_positive <-> DCM Status Channel 2/Status/Moving positive
//     PlcTask Inputs/GVL_iXlinker.EtherCAT_Master_EPPxxxx.Beckhoff_EPP7xxx.Beckhoff_EPP7xxxEK1122.A_0009_EPP7342_0002_0017.DCM_Status_Channel_1.Status/Moving_negative <-> DCM Status Channel 1/Status/Moving negative
//     PlcTask Inputs/GVL_iXlinker.EtherCAT_Master_EPPxxxx.Beckhoff_EPP7xxx.Beckhoff_EPP7xxxEK1122.A_0009_EPP7342_0002_0017.DCM_Status_Channel_2.Status/Moving_negative <-> DCM Status Channel 2/Status/Moving negative
//     PlcTask Inputs/GVL_iXlinker.EtherCAT_Master_EPPxxxx.Beckhoff_EPP7xxx.Beckhoff_EPP7xxxEK1122.A_0009_EPP7342_0002_0017.DCM_Status_Channel_1.Status/Torque_reduced <-> DCM Status Channel 1/Status/Torque reduced
//     PlcTask Inputs/GVL_iXlinker.EtherCAT_Master_EPPxxxx.Beckhoff_EPP7xxx.Beckhoff_EPP7xxxEK1122.A_0009_EPP7342_0002_0017.DCM_Status_Channel_2.Status/Torque_reduced <-> DCM Status Channel 2/Status/Torque reduced
//     PlcTask Inputs/GVL_iXlinker.EtherCAT_Master_EPPxxxx.Beckhoff_EPP7xxx.Beckhoff_EPP7xxxEK1122.A_0009_EPP7342_0002_0017.DCM_Status_Channel_1.Status/Digital_input_1 <-> DCM Status Channel 1/Status/Digital input 1
//     PlcTask Inputs/GVL_iXlinker.EtherCAT_Master_EPPxxxx.Beckhoff_EPP7xxx.Beckhoff_EPP7xxxEK1122.A_0009_EPP7342_0002_0017.DCM_Status_Channel_1.Status/Digital_input_2 <-> DCM Status Channel 1/Status/Digital input 2
//     PlcTask Inputs/GVL_iXlinker.EtherCAT_Master_EPPxxxx.Beckhoff_EPP7xxx.Beckhoff_EPP7xxxEK1122.A_0009_EPP7342_0002_0017.DCM_Status_Channel_2.Status/Digital_input_1 <-> DCM Status Channel 2/Status/Digital input 1
//     PlcTask Inputs/GVL_iXlinker.EtherCAT_Master_EPPxxxx.Beckhoff_EPP7xxx.Beckhoff_EPP7xxxEK1122.A_0009_EPP7342_0002_0017.DCM_Status_Channel_2.Status/Digital_input_2 <-> DCM Status Channel 2/Status/Digital input 2
//     PlcTask Inputs/GVL_iXlinker.EtherCAT_Master_EPPxxxx.Beckhoff_EPP7xxx.Beckhoff_EPP7xxxEK1122.A_0009_EPP7342_0002_0017.DCM_Status_Channel_1.Status/Sync_error <-> DCM Status Channel 1/Status/Sync error
//     PlcTask Inputs/GVL_iXlinker.EtherCAT_Master_EPPxxxx.Beckhoff_EPP7xxx.Beckhoff_EPP7xxxEK1122.A_0009_EPP7342_0002_0017.DCM_Status_Channel_2.Status/Sync_error <-> DCM Status Channel 2/Status/Sync error
//     PlcTask Inputs/GVL_iXlinker.EtherCAT_Master_EPPxxxx.Beckhoff_EPP7xxx.Beckhoff_EPP7xxxEK1122.A_0009_EPP7342_0002_0017.DCM_Status_Channel_1.Status/TxPDO_Toggle <-> DCM Status Channel 1/Status/TxPDO Toggle
//     PlcTask Inputs/GVL_iXlinker.EtherCAT_Master_EPPxxxx.Beckhoff_EPP7xxx.Beckhoff_EPP7xxxEK1122.A_0009_EPP7342_0002_0017.DCM_Status_Channel_2.Status/TxPDO_Toggle <-> DCM Status Channel 2/Status/TxPDO Toggle
//     PlcTask Outputs/GVL_iXlinker.EtherCAT_Master_EPPxxxx.Beckhoff_EPP7xxx.Beckhoff_EPP7xxxEK1122.A_0009_EPP7342_0002_0017.ENC_Control_compact_Channel_1.Control/Enable_latch_extern_on_positive_edge <-> ENC Control compact Channel 1/Control/Enable latch extern on positive edge
//     PlcTask Outputs/GVL_iXlinker.EtherCAT_Master_EPPxxxx.Beckhoff_EPP7xxx.Beckhoff_EPP7xxxEK1122.A_0009_EPP7342_0002_0017.ENC_Control_compact_Channel_2.Control/Enable_latch_extern_on_positive_edge <-> ENC Control compact Channel 2/Control/Enable latch extern on positive edge
//     PlcTask Outputs/GVL_iXlinker.EtherCAT_Master_EPPxxxx.Beckhoff_EPP7xxx.Beckhoff_EPP7xxxEK1122.A_0009_EPP7342_0002_0017.ENC_Control_compact_Channel_1.Control/Set_counter <-> ENC Control compact Channel 1/Control/Set counter
//     PlcTask Outputs/GVL_iXlinker.EtherCAT_Master_EPPxxxx.Beckhoff_EPP7xxx.Beckhoff_EPP7xxxEK1122.A_0009_EPP7342_0002_0017.ENC_Control_compact_Channel_2.Control/Set_counter <-> ENC Control compact Channel 2/Control/Set counter
//     PlcTask Outputs/GVL_iXlinker.EtherCAT_Master_EPPxxxx.Beckhoff_EPP7xxx.Beckhoff_EPP7xxxEK1122.A_0009_EPP7342_0002_0017.ENC_Control_compact_Channel_1.Control/Enable_latch_extern_on_negative_edge <-> ENC Control compact Channel 1/Control/Enable latch extern on negative edge
//     PlcTask Outputs/GVL_iXlinker.EtherCAT_Master_EPPxxxx.Beckhoff_EPP7xxx.Beckhoff_EPP7xxxEK1122.A_0009_EPP7342_0002_0017.ENC_Control_compact_Channel_2.Control/Enable_latch_extern_on_negative_edge <-> ENC Control compact Channel 2/Control/Enable latch extern on negative edge
//     PlcTask Outputs/GVL_iXlinker.EtherCAT_Master_EPPxxxx.Beckhoff_EPP7xxx.Beckhoff_EPP7xxxEK1122.A_0009_EPP7342_0002_0017.ENC_Control_compact_Channel_1.Set_counter_value <-> ENC Control compact Channel 1/Set counter value
//     PlcTask Outputs/GVL_iXlinker.EtherCAT_Master_EPPxxxx.Beckhoff_EPP7xxx.Beckhoff_EPP7xxxEK1122.A_0009_EPP7342_0002_0017.ENC_Control_compact_Channel_2.Set_counter_value <-> ENC Control compact Channel 2/Set counter value
//     PlcTask Outputs/GVL_iXlinker.EtherCAT_Master_EPPxxxx.Beckhoff_EPP7xxx.Beckhoff_EPP7xxxEK1122.A_0009_EPP7342_0002_0017.DCM_Control_Channel_1.Control/Enable <-> DCM Control Channel 1/Control/Enable
//     PlcTask Outputs/GVL_iXlinker.EtherCAT_Master_EPPxxxx.Beckhoff_EPP7xxx.Beckhoff_EPP7xxxEK1122.A_0009_EPP7342_0002_0017.DCM_Control_Channel_2.Control/Enable <-> DCM Control Channel 2/Control/Enable
//     PlcTask Outputs/GVL_iXlinker.EtherCAT_Master_EPPxxxx.Beckhoff_EPP7xxx.Beckhoff_EPP7xxxEK1122.A_0009_EPP7342_0002_0017.DCM_Control_Channel_1.Control/Reset <-> DCM Control Channel 1/Control/Reset
//     PlcTask Outputs/GVL_iXlinker.EtherCAT_Master_EPPxxxx.Beckhoff_EPP7xxx.Beckhoff_EPP7xxxEK1122.A_0009_EPP7342_0002_0017.DCM_Control_Channel_2.Control/Reset <-> DCM Control Channel 2/Control/Reset
//     PlcTask Outputs/GVL_iXlinker.EtherCAT_Master_EPPxxxx.Beckhoff_EPP7xxx.Beckhoff_EPP7xxxEK1122.A_0009_EPP7342_0002_0017.DCM_Control_Channel_1.Control/Reduce_torque <-> DCM Control Channel 1/Control/Reduce torque
//     PlcTask Outputs/GVL_iXlinker.EtherCAT_Master_EPPxxxx.Beckhoff_EPP7xxx.Beckhoff_EPP7xxxEK1122.A_0009_EPP7342_0002_0017.DCM_Control_Channel_2.Control/Reduce_torque <-> DCM Control Channel 2/Control/Reduce torque
//     PlcTask Outputs/GVL_iXlinker.EtherCAT_Master_EPPxxxx.Beckhoff_EPP7xxx.Beckhoff_EPP7xxxEK1122.A_0009_EPP7342_0002_0017.DCM_Velocity_Channel_1.Velocity <-> DCM Velocity Channel 1/Velocity
//     PlcTask Outputs/GVL_iXlinker.EtherCAT_Master_EPPxxxx.Beckhoff_EPP7xxx.Beckhoff_EPP7xxxEK1122.A_0009_EPP7342_0002_0017.DCM_Velocity_Channel_2.Velocity <-> DCM Velocity Channel 2/Velocity
//     PlcTask Inputs/GVL_iXlinker.EtherCAT_Master_EPPxxxx.Beckhoff_EPP7xxx.Beckhoff_EPP7xxxEK1122.A_0009_EPP7342_0002_0017.WcState.WcState <-> WcState/WcState
//     PlcTask Inputs/GVL_iXlinker.EtherCAT_Master_EPPxxxx.Beckhoff_EPP7xxx.Beckhoff_EPP7xxxEK1122.A_0009_EPP7342_0002_0017.WcState.InputToggle <-> WcState/InputToggle
//     PlcTask Inputs/GVL_iXlinker.EtherCAT_Master_EPPxxxx.Beckhoff_EPP7xxx.Beckhoff_EPP7xxxEK1122.A_0009_EPP7342_0002_0017.InfoData.AdsAddr <-> InfoData/AdsAddr
//     PlcTask Inputs/GVL_iXlinker.EtherCAT_Master_EPPxxxx.Beckhoff_EPP7xxx.Beckhoff_EPP7xxxEK1122.A_0009_EPP7342_0002_0017.InfoData.Chn0 <-> InfoData/Chn0
//     PlcTask Inputs/GVL_iXlinker.EtherCAT_Master_EPPxxxx.Beckhoff_EPP7xxx.Beckhoff_EPP7xxxEK1122.A_0009_EPP7342_0002_0017.InfoData.Chn1 <-> InfoData/Chn1
//     PlcTask Inputs/GVL_iXlinker.EtherCAT_Master_EPPxxxx.Beckhoff_EPP7xxx.Beckhoff_EPP7xxxEK1122.A_0009_EPP7342_0002_0017.InfoData.Chn2 <-> InfoData/Chn2
//     PlcTask Inputs/GVL_iXlinker.EtherCAT_Master_EPPxxxx.Beckhoff_EPP7xxx.Beckhoff_EPP7xxxEK1122.A_0009_EPP7342_0002_0017.InfoData.Chn3 <-> InfoData/Chn3
//     PlcTask Inputs/GVL_iXlinker.EtherCAT_Master_EPPxxxx.Beckhoff_EPP7xxx.Beckhoff_EPP7xxxEK1122.A_0009_EPP7342_0002_0017.InfoData.State <-> InfoData/State
//   PLC/PLC Instance <-> EtherCAT Master EPPxxxx/Beckhoff EPP9xxx
//     PlcTask Inputs/GVL_iXlinker.EtherCAT_Master_EPPxxxx.Beckhoff_EPP9xxx.InfoData.State <-> InfoData/State
//   PLC/PLC Instance <-> EtherCAT Master EPPxxxx/Beckhoff EPP9xxx/Beckhoff EPP9xxxEK1122
//     PlcTask Inputs/GVL_iXlinker.EtherCAT_Master_EPPxxxx.Beckhoff_EPP9xxx.Beckhoff_EPP9xxxEK1122.InfoData.State <-> InfoData/State
//   PLC/PLC Instance <-> EtherCAT Master EPPxxxx/Beckhoff EPP9xxx/Beckhoff EPP9xxxEK1122/Beckhoff EPP9xxxsub EK1100
//     PlcTask Inputs/GVL_iXlinker.EtherCAT_Master_EPPxxxx.Beckhoff_EPP9xxx.Beckhoff_EPP9xxxEK1122.Beckhoff_EPP9xxxsub_EK1100.InfoData.State <-> InfoData/State
//   PLC/PLC Instance <-> EtherCAT Master EPPxxxx/Beckhoff EPP9xxx/Beckhoff EPP9xxxEK1122/A_0001(EPP9001-0060-0016)
//     PlcTask Inputs/GVL_iXlinker.EtherCAT_Master_EPPxxxx.Beckhoff_EPP9xxx.Beckhoff_EPP9xxxEK1122.A_0001_EPP9001_0060_0016.InfoData.State <-> InfoData/State
//   PLC/PLC Instance <-> EtherCAT Master EPPxxxx/Beckhoff EPP9xxx/Beckhoff EPP9xxxEK1122/A_0002(EPP9001-0060-0017)
//     PlcTask Inputs/GVL_iXlinker.EtherCAT_Master_EPPxxxx.Beckhoff_EPP9xxx.Beckhoff_EPP9xxxEK1122.A_0002_EPP9001_0060_0017.InfoData.State <-> InfoData/State
//   PLC/PLC Instance <-> EtherCAT Master EPPxxxx/Beckhoff EPP9xxx/Beckhoff EPP9xxxEK1122/A_0003(EPP9022-0060-0017)
//     PlcTask Inputs/GVL_iXlinker.EtherCAT_Master_EPPxxxx.Beckhoff_EPP9xxx.Beckhoff_EPP9xxxEK1122.A_0003_EPP9022_0060_0017.EPM_Inputs_Channel_1.Status/Voltage_min_error <-> EPM Inputs Channel 1/Status/Voltage min error
//     PlcTask Inputs/GVL_iXlinker.EtherCAT_Master_EPPxxxx.Beckhoff_EPP9xxx.Beckhoff_EPP9xxxEK1122.A_0003_EPP9022_0060_0017.EPM_Inputs_Channel_2.Status/Voltage_min_error <-> EPM Inputs Channel 2/Status/Voltage min error
//     PlcTask Inputs/GVL_iXlinker.EtherCAT_Master_EPPxxxx.Beckhoff_EPP9xxx.Beckhoff_EPP9xxxEK1122.A_0003_EPP9022_0060_0017.EPM_Inputs_Channel_1.Status/Voltage_max_error <-> EPM Inputs Channel 1/Status/Voltage max error
//     PlcTask Inputs/GVL_iXlinker.EtherCAT_Master_EPPxxxx.Beckhoff_EPP9xxx.Beckhoff_EPP9xxxEK1122.A_0003_EPP9022_0060_0017.EPM_Inputs_Channel_2.Status/Voltage_max_error <-> EPM Inputs Channel 2/Status/Voltage max error
//     PlcTask Inputs/GVL_iXlinker.EtherCAT_Master_EPPxxxx.Beckhoff_EPP9xxx.Beckhoff_EPP9xxxEK1122.A_0003_EPP9022_0060_0017.EPM_Inputs_Channel_1.Status/Current_max_error <-> EPM Inputs Channel 1/Status/Current max error
//     PlcTask Inputs/GVL_iXlinker.EtherCAT_Master_EPPxxxx.Beckhoff_EPP9xxx.Beckhoff_EPP9xxxEK1122.A_0003_EPP9022_0060_0017.EPM_Inputs_Channel_2.Status/Current_max_error <-> EPM Inputs Channel 2/Status/Current max error
//     PlcTask Inputs/GVL_iXlinker.EtherCAT_Master_EPPxxxx.Beckhoff_EPP9xxx.Beckhoff_EPP9xxxEK1122.A_0003_EPP9022_0060_0017.EPM_Inputs_Channel_1.Status/Voltage_min_warning <-> EPM Inputs Channel 1/Status/Voltage min warning
//     PlcTask Inputs/GVL_iXlinker.EtherCAT_Master_EPPxxxx.Beckhoff_EPP9xxx.Beckhoff_EPP9xxxEK1122.A_0003_EPP9022_0060_0017.EPM_Inputs_Channel_2.Status/Voltage_min_warning <-> EPM Inputs Channel 2/Status/Voltage min warning
//     PlcTask Inputs/GVL_iXlinker.EtherCAT_Master_EPPxxxx.Beckhoff_EPP9xxx.Beckhoff_EPP9xxxEK1122.A_0003_EPP9022_0060_0017.EPM_Inputs_Channel_1.Status/Voltage_max_warning <-> EPM Inputs Channel 1/Status/Voltage max warning
//     PlcTask Inputs/GVL_iXlinker.EtherCAT_Master_EPPxxxx.Beckhoff_EPP9xxx.Beckhoff_EPP9xxxEK1122.A_0003_EPP9022_0060_0017.EPM_Inputs_Channel_2.Status/Voltage_max_warning <-> EPM Inputs Channel 2/Status/Voltage max warning
//     PlcTask Inputs/GVL_iXlinker.EtherCAT_Master_EPPxxxx.Beckhoff_EPP9xxx.Beckhoff_EPP9xxxEK1122.A_0003_EPP9022_0060_0017.EPM_Inputs_Channel_1.Status/Current_max_warning <-> EPM Inputs Channel 1/Status/Current max warning
//     PlcTask Inputs/GVL_iXlinker.EtherCAT_Master_EPPxxxx.Beckhoff_EPP9xxx.Beckhoff_EPP9xxxEK1122.A_0003_EPP9022_0060_0017.EPM_Inputs_Channel_2.Status/Current_max_warning <-> EPM Inputs Channel 2/Status/Current max warning
//     PlcTask Inputs/GVL_iXlinker.EtherCAT_Master_EPPxxxx.Beckhoff_EPP9xxx.Beckhoff_EPP9xxxEK1122.A_0003_EPP9022_0060_0017.EPM_Inputs_Channel_1.Status/Channel_error <-> EPM Inputs Channel 1/Status/Channel error
//     PlcTask Inputs/GVL_iXlinker.EtherCAT_Master_EPPxxxx.Beckhoff_EPP9xxx.Beckhoff_EPP9xxxEK1122.A_0003_EPP9022_0060_0017.EPM_Inputs_Channel_2.Status/Channel_error <-> EPM Inputs Channel 2/Status/Channel error
//     PlcTask Inputs/GVL_iXlinker.EtherCAT_Master_EPPxxxx.Beckhoff_EPP9xxx.Beckhoff_EPP9xxxEK1122.A_0003_EPP9022_0060_0017.EPM_Inputs_Channel_1.Status/Channel_warning <-> EPM Inputs Channel 1/Status/Channel warning
//     PlcTask Inputs/GVL_iXlinker.EtherCAT_Master_EPPxxxx.Beckhoff_EPP9xxx.Beckhoff_EPP9xxxEK1122.A_0003_EPP9022_0060_0017.EPM_Inputs_Channel_2.Status/Channel_warning <-> EPM Inputs Channel 2/Status/Channel warning
//     PlcTask Inputs/GVL_iXlinker.EtherCAT_Master_EPPxxxx.Beckhoff_EPP9xxx.Beckhoff_EPP9xxxEK1122.A_0003_EPP9022_0060_0017.EPM_Inputs_Channel_1.Status/TxPDO_State <-> EPM Inputs Channel 1/Status/TxPDO State
//     PlcTask Inputs/GVL_iXlinker.EtherCAT_Master_EPPxxxx.Beckhoff_EPP9xxx.Beckhoff_EPP9xxxEK1122.A_0003_EPP9022_0060_0017.EPM_Inputs_Channel_2.Status/TxPDO_State <-> EPM Inputs Channel 2/Status/TxPDO State
//     PlcTask Inputs/GVL_iXlinker.EtherCAT_Master_EPPxxxx.Beckhoff_EPP9xxx.Beckhoff_EPP9xxxEK1122.A_0003_EPP9022_0060_0017.EPM_Inputs_Channel_1.Status/TxPDO_Toggle <-> EPM Inputs Channel 1/Status/TxPDO Toggle
//     PlcTask Inputs/GVL_iXlinker.EtherCAT_Master_EPPxxxx.Beckhoff_EPP9xxx.Beckhoff_EPP9xxxEK1122.A_0003_EPP9022_0060_0017.EPM_Inputs_Channel_2.Status/TxPDO_Toggle <-> EPM Inputs Channel 2/Status/TxPDO Toggle
